      A(    ;
      A     M   1000.5;
      A     DB51.DBX  204.3;
      A     DB51.DBX  203.7;
      AN    DB51.DBX  203.6;
      O     ;
      A     M   1000.6;
      AN    M   1001.0;
      A     M   1100.1;
      O     M   1001.2;
      )     ;
      A     M   1103.1;
      AN    M   1101.7;
      AN    Q    236.6;
      =     Q    236.7;
NETWORK
TITLE =

      A(    ;
      A     M   1000.5;
      A     DB51.DBX  204.4;
      A     DB51.DBX  203.6;
      AN    DB51.DBX  203.7;
      O     ;
      A     M   1000.6;
      AN    M   1001.0;
      A     M   1100.0;
      A     M   5016.0;
      )     ;
      A     M   1103.3;
      AN    M   1102.0;
      AN    Q    237.1;
      =     Q    237.0;
NETWORK
TITLE =

      A(    ;
      A     M   1000.5;
      A     DB51.DBX  204.4;
      A     DB51.DBX  203.7;
      AN    DB51.DBX  203.6;
      O     ;
      A     M   1000.6;
      AN    M   1001.0;
      A     M   1100.1;
      O     M   1001.2;
      )     ;
      A     M   1103.3;
      AN    M   1102.1;
      AN    Q    237.0;
      =     Q    237.1;
NETWORK
TITLE =

      A(    ;
      A     M   1000.5;
      A     DB51.DBX  204.5;
      A     DB51.DBX  203.6;
      AN    DB51.DBX  203.7;
      O     ;
      A     M   1000.6;
      AN    M   1001.0;
      A     M   1100.0;
      A     M   5016.0;
      )     ;
      AN    M   1102.2;
      AN    Q    237.3;
      =     Q    237.2;
NETWORK
TITLE =

      A(    ;
      A     M   1000.5;
      A     DB51.DBX  204.5;
      A     DB51.DBX  203.7;
      AN    DB51.DBX  203.6;
      O     ;
      A     M   1000.6;
      AN    M   1001.0;
      A     M   1100.1;
      A     M   1106.3;
      O     M   1001.2;
      )     ;
      AN    M   1102.3;
      AN    Q    237.2;
      =     Q    237.3;
NETWORK
TITLE =
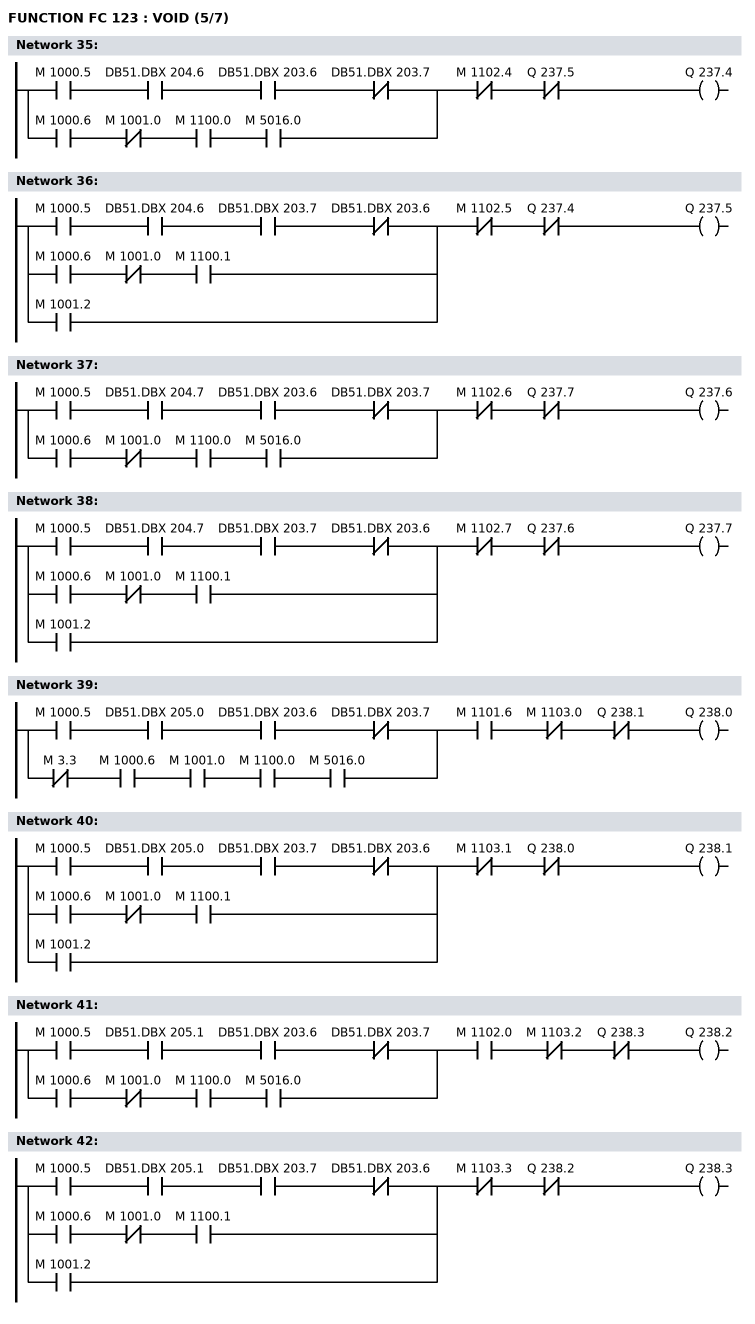

      A(    ;
      A     M   1000.5;
      A     DB51.DBX  204.6;
      A     DB51.DBX  203.6;
      AN    DB51.DBX  203.7;
      O     ;
      A     M   1000.6;
      AN    M   1001.0;
      A     M   1100.0;
      A     M   5016.0;
      )     ;
      AN    M   1102.4;
      AN    Q    237.5;
      =     Q    237.4;
NETWORK
TITLE =

      A(    ;
      A     M   1000.5;
      A     DB51.DBX  204.6;
      A     DB51.DBX  203.7;
      AN    DB51.DBX  203.6;
      O     ;
      A     M   1000.6;
      AN    M   1001.0;
      A     M   1100.1;
      O     M   1001.2;
      )     ;
      AN    M   1102.5;
      AN    Q    237.4;
      =     Q    237.5;
NETWORK
TITLE =

      A(    ;
      A     M   1000.5;
      A     DB51.DBX  204.7;
      A     DB51.DBX  203.6;
      AN    DB51.DBX  203.7;
      O     ;
      A     M   1000.6;
      AN    M   1001.0;
      A     M   1100.0;
      A     M   5016.0;
      )     ;
      AN    M   1102.6;
      AN    Q    237.7;
      =     Q    237.6;
NETWORK
TITLE =

      A(    ;
      A     M   1000.5;
      A     DB51.DBX  204.7;
      A     DB51.DBX  203.7;
      AN    DB51.DBX  203.6;
      O     ;
      A     M   1000.6;
      AN    M   1001.0;
      A     M   1100.1;
      O     M   1001.2;
      )     ;
      AN    M   1102.7;
      AN    Q    237.6;
      =     Q    237.7;
NETWORK
TITLE =

      A(    ;
      A     M   1000.5;
      A     DB51.DBX  205.0;
      A     DB51.DBX  203.6;
      AN    DB51.DBX  203.7;
      O     ;
      AN    M      3.3;
      A     M   1000.6;
      A     M   1001.0;
      A     M   1100.0;
      A     M   5016.0;
      )     ;
      A     M   1101.6;
      AN    M   1103.0;
      AN    Q    238.1;
      =     Q    238.0;
NETWORK
TITLE =

      A(    ;
      A     M   1000.5;
      A     DB51.DBX  205.0;
      A     DB51.DBX  203.7;
      AN    DB51.DBX  203.6;
      O     ;
      A     M   1000.6;
      AN    M   1001.0;
      A     M   1100.1;
      O     M   1001.2;
      )     ;
      AN    M   1103.1;
      AN    Q    238.0;
      =     Q    238.1;
NETWORK
TITLE =

      A(    ;
      A     M   1000.5;
      A     DB51.DBX  205.1;
      A     DB51.DBX  203.6;
      AN    DB51.DBX  203.7;
      O     ;
      A     M   1000.6;
      AN    M   1001.0;
      A     M   1100.0;
      A     M   5016.0;
      )     ;
      A     M   1102.0;
      AN    M   1103.2;
      AN    Q    238.3;
      =     Q    238.2;
NETWORK
TITLE =

      A(    ;
      A     M   1000.5;
      A     DB51.DBX  205.1;
      A     DB51.DBX  203.7;
      AN    DB51.DBX  203.6;
      O     ;
      A     M   1000.6;
      AN    M   1001.0;
      A     M   1100.1;
      O     M   1001.2;
      )     ;
      AN    M   1103.3;
      AN    Q    238.2;
      =     Q    238.3;
NETWORK
TITLE =
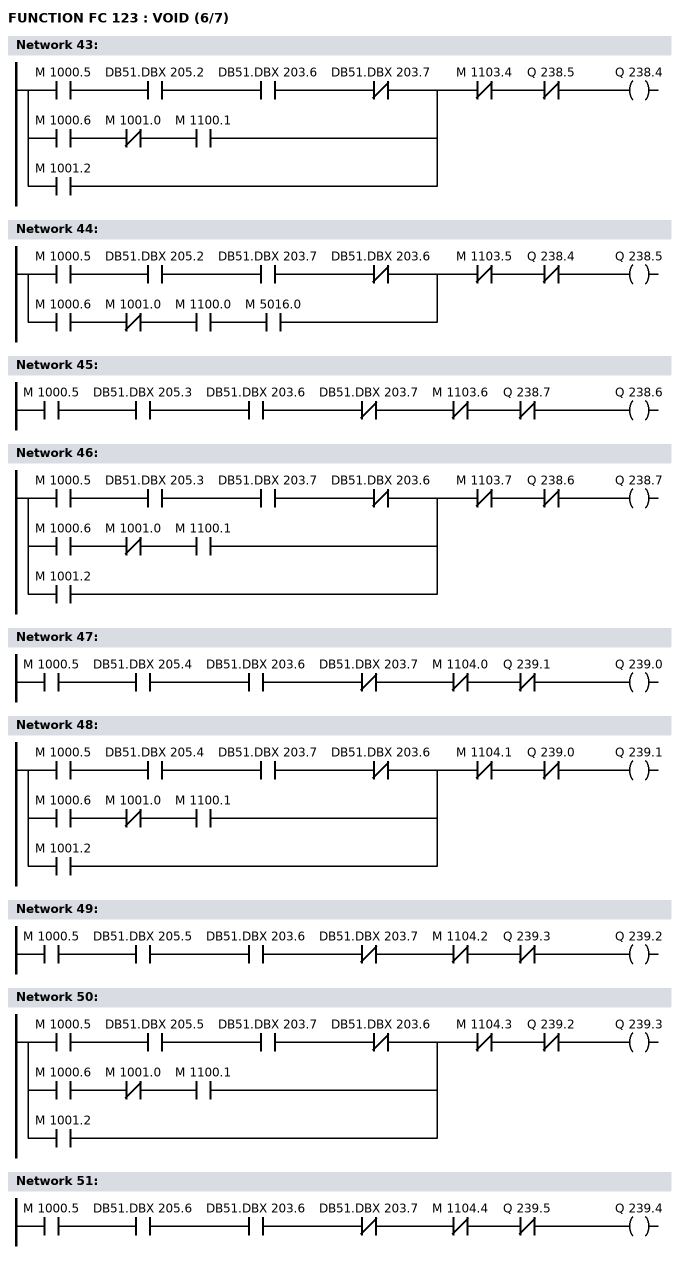

      A(    ;
      A     M   1000.5;
      A     DB51.DBX  205.2;
      A     DB51.DBX  203.6;
      AN    DB51.DBX  203.7;
      O     ;
      A     M   1000.6;
      AN    M   1001.0;
      A     M   1100.1;
      O     M   1001.2;
      )     ;
      AN    M   1103.4;
      AN    Q    238.5;
      =     Q    238.4;
NETWORK
TITLE =

      A(    ;
      A     M   1000.5;
      A     DB51.DBX  205.2;
      A     DB51.DBX  203.7;
      AN    DB51.DBX  203.6;
      O     ;
      A     M   1000.6;
      AN    M   1001.0;
      A     M   1100.0;
      A     M   5016.0;
      )     ;
      AN    M   1103.5;
      AN    Q    238.4;
      =     Q    238.5;
NETWORK
TITLE =

      A     M   1000.5;
      A     DB51.DBX  205.3;
      A     DB51.DBX  203.6;
      AN    DB51.DBX  203.7;
      AN    M   1103.6;
      AN    Q    238.7;
      =     Q    238.6;
NETWORK
TITLE =

      A(    ;
      A     M   1000.5;
      A     DB51.DBX  205.3;
      A     DB51.DBX  203.7;
      AN    DB51.DBX  203.6;
      O     ;
      A     M   1000.6;
      AN    M   1001.0;
      A     M   1100.1;
      O     M   1001.2;
      )     ;
      AN    M   1103.7;
      AN    Q    238.6;
      =     Q    238.7;
NETWORK
TITLE =

      A     M   1000.5;
      A     DB51.DBX  205.4;
      A     DB51.DBX  203.6;
      AN    DB51.DBX  203.7;
      AN    M   1104.0;
      AN    Q    239.1;
      =     Q    239.0;
NETWORK
TITLE =

      A(    ;
      A     M   1000.5;
      A     DB51.DBX  205.4;
      A     DB51.DBX  203.7;
      AN    DB51.DBX  203.6;
      O     ;
      A     M   1000.6;
      AN    M   1001.0;
      A     M   1100.1;
      O     M   1001.2;
      )     ;
      AN    M   1104.1;
      AN    Q    239.0;
      =     Q    239.1;
NETWORK
TITLE =

      A     M   1000.5;
      A     DB51.DBX  205.5;
      A     DB51.DBX  203.6;
      AN    DB51.DBX  203.7;
      AN    M   1104.2;
      AN    Q    239.3;
      =     Q    239.2;
NETWORK
TITLE =

      A(    ;
      A     M   1000.5;
      A     DB51.DBX  205.5;
      A     DB51.DBX  203.7;
      AN    DB51.DBX  203.6;
      O     ;
      A     M   1000.6;
      AN    M   1001.0;
      A     M   1100.1;
      O     M   1001.2;
      )     ;
      AN    M   1104.3;
      AN    Q    239.2;
      =     Q    239.3;
NETWORK
TITLE =

      A     M   1000.5;
      A     DB51.DBX  205.6;
      A     DB51.DBX  203.6;
      AN    DB51.DBX  203.7;
      AN    M   1104.4;
      AN    Q    239.5;
      =     Q    239.4;
NETWORK
TITLE =
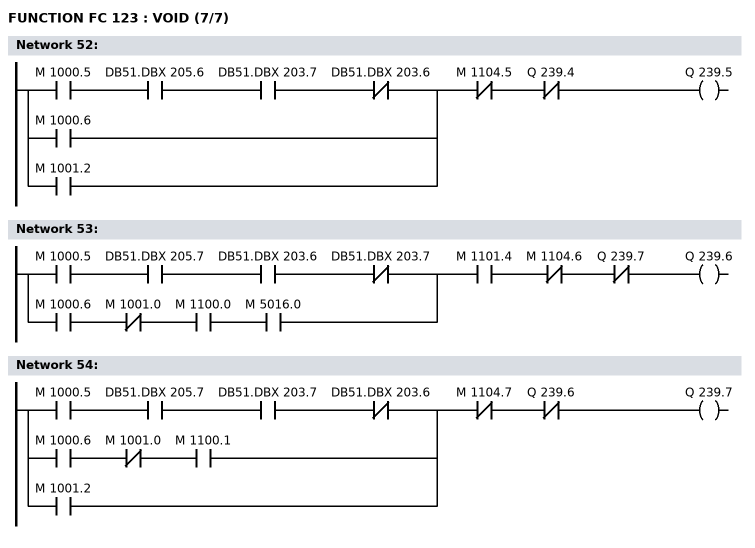

      A(    ;
      A     M   1000.5;
      A     DB51.DBX  205.6;
      A     DB51.DBX  203.7;
      AN    DB51.DBX  203.6;
      O     M   1000.6;
      O     M   1001.2;
      )     ;
      AN    M   1104.5;
      AN    Q    239.4;
      =     Q    239.5;
NETWORK
TITLE =

      A(    ;
      A     M   1000.5;
      A     DB51.DBX  205.7;
      A     DB51.DBX  203.6;
      AN    DB51.DBX  203.7;
      O     ;
      A     M   1000.6;
      AN    M   1001.0;
      A     M   1100.0;
      A     M   5016.0;
      )     ;
      A     M   1101.4;
      AN    M   1104.6;
      AN    Q    239.7;
      =     Q    239.6;
NETWORK
TITLE =

      A(    ;
      A     M   1000.5;
      A     DB51.DBX  205.7;
      A     DB51.DBX  203.7;
      AN    DB51.DBX  203.6;
      O     ;
      A     M   1000.6;
      AN    M   1001.0;
      A     M   1100.1;
      O     M   1001.2;
      )     ;
      AN    M   1104.7;
      AN    Q    239.6;
      =     Q    239.7;
END_FUNCTION

FUNCTION_BLOCK FB 124
TITLE =
VERSION : 0.1


VAR
  S702_TL_DC_PIN : FB 426;
  S702_TL_DC_LATCH1 : FB 426;
  S702_TL_DC_LATCH2 : FB 426;
  S702_TL_DC_1ST_CLAMP1 : FB 426;
  S702_TL_DC_1ST_CLAMP2 : FB 426;
  S702_TL_DC_1ST_CLAMP3 : FB 426;
  S702_TL_DC_2ND_CLAMP1 : FB 426;
  S702_TL_DC_2ND_CLAMP2 : FB 426;
  S702_TL_DC_U261 : FB 426;
  S702_TL_DC_U261_CLAMP : FB 426;
  S702_TL_DC_U269 : FB 426;
  S702_TL_DC_U269_CLAMP : FB 426;
  S702_TL_DC_3RD_CLAMP : FB 426;
  S702_TL_DC_U262_1_UP_DN : FB 426;
  S702_TL_DC_U262_1 : FB 426;
  S702_TL_DC_U262_1_CLAMP : FB 426;
  S702_TL_DC_U261_2_CLAMP : FB 426;
END_VAR
BEGIN
NETWORK
TITLE =
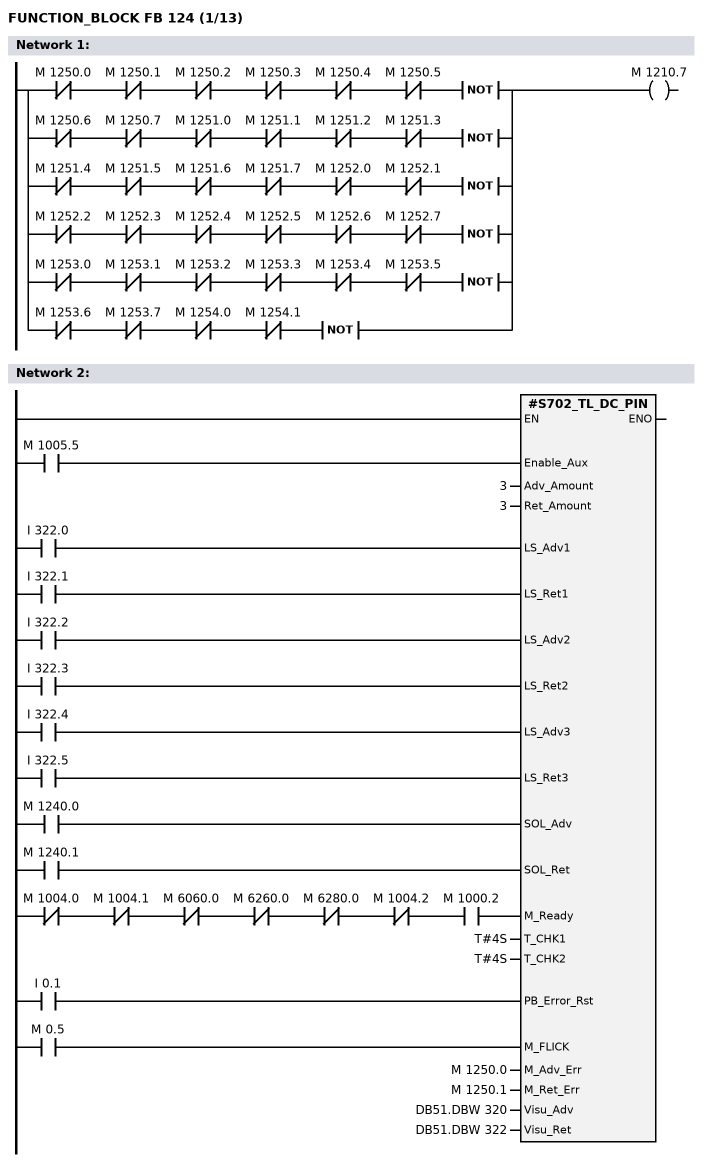

      AN    M   1250.0;
      AN    M   1250.1;
      AN    M   1250.2;
      AN    M   1250.3;
      AN    M   1250.4;
      AN    M   1250.5;
      NOT   ;
      O(    ;
      AN    M   1250.6;
      AN    M   1250.7;
      AN    M   1251.0;
      AN    M   1251.1;
      AN    M   1251.2;
      AN    M   1251.3;
      NOT   ;
      )     ;
      O(    ;
      AN    M   1251.4;
      AN    M   1251.5;
      AN    M   1251.6;
      AN    M   1251.7;
      AN    M   1252.0;
      AN    M   1252.1;
      NOT   ;
      )     ;
      O(    ;
      AN    M   1252.2;
      AN    M   1252.3;
      AN    M   1252.4;
      AN    M   1252.5;
      AN    M   1252.6;
      AN    M   1252.7;
      NOT   ;
      )     ;
      O(    ;
      AN    M   1253.0;
      AN    M   1253.1;
      AN    M   1253.2;
      AN    M   1253.3;
      AN    M   1253.4;
      AN    M   1253.5;
      NOT   ;
      )     ;
      O(    ;
      AN    M   1253.6;
      AN    M   1253.7;
      AN    M   1254.0;
      AN    M   1254.1;
      NOT   ;
      )     ;
      =     M   1210.7;
NETWORK
TITLE =

      A     M   1005.5;
      =     L      0.0;
      BLD   103;
      A     I    322.0;
      =     L      0.1;
      BLD   103;
      A     I    322.1;
      =     L      0.2;
      BLD   103;
      A     I    322.2;
      =     L      0.3;
      BLD   103;
      A     I    322.3;
      =     L      0.4;
      BLD   103;
      A     I    322.4;
      =     L      0.5;
      BLD   103;
      A     I    322.5;
      =     L      0.6;
      BLD   103;
      A     M   1240.0;
      =     L      2.1;
      BLD   103;
      A     M   1240.1;
      =     L      2.2;
      BLD   103;
      AN    M   1004.0;
      AN    M   1004.1;
      AN    M   6060.0;
      AN    M   6260.0;
      AN    M   6280.0;
      AN    M   1004.2;
      A     M   1000.2;
      =     L      2.3;
      BLD   103;
      A     I      0.1;
      =     L      2.5;
      BLD   103;
      A     M      0.5;
      =     L      2.6;
      BLD   103;
      CALL #S702_TL_DC_PIN (
           Enable_Aux               := L      0.0,
           Adv_Amount               := 3,
           Ret_Amount               := 3,
           LS_Adv1                  := L      0.1,
           LS_Ret1                  := L      0.2,
           LS_Adv2                  := L      0.3,
           LS_Ret2                  := L      0.4,
           LS_Adv3                  := L      0.5,
           LS_Ret3                  := L      0.6,
           SOL_Adv                  := L      2.1,
           SOL_Ret                  := L      2.2,
           M_Ready                  := L      2.3,
           T_CHK1                   := T#4S,
           T_CHK2                   := T#4S,
           PB_Error_Rst             := L      2.5,
           M_FLICK                  := L      2.6,
           M_Adv_Err                := M   1250.0,
           M_Ret_Err                := M   1250.1,
           Visu_Adv                 := DB51.DBW  320,
           Visu_Ret                 := DB51.DBW  322);
      NOP   0;
NETWORK
TITLE =
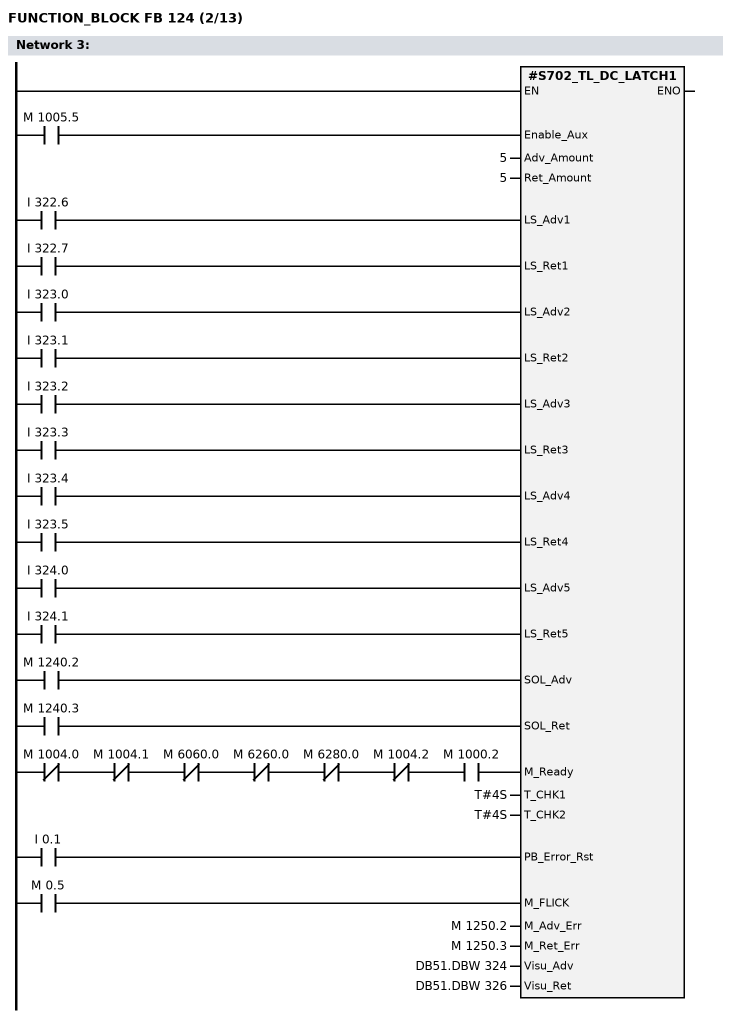

      A     M   1005.5;
      =     L      0.0;
      BLD   103;
      A     I    322.6;
      =     L      0.1;
      BLD   103;
      A     I    322.7;
      =     L      0.2;
      BLD   103;
      A     I    323.0;
      =     L      0.3;
      BLD   103;
      A     I    323.1;
      =     L      0.4;
      BLD   103;
      A     I    323.2;
      =     L      0.5;
      BLD   103;
      A     I    323.3;
      =     L      0.6;
      BLD   103;
      A     I    323.4;
      =     L      0.7;
      BLD   103;
      A     I    323.5;
      =     L      1.0;
      BLD   103;
      A     I    324.0;
      =     L      1.1;
      BLD   103;
      A     I    324.1;
      =     L      1.2;
      BLD   103;
      A     M   1240.2;
      =     L      2.1;
      BLD   103;
      A     M   1240.3;
      =     L      2.2;
      BLD   103;
      AN    M   1004.0;
      AN    M   1004.1;
      AN    M   6060.0;
      AN    M   6260.0;
      AN    M   6280.0;
      AN    M   1004.2;
      A     M   1000.2;
      =     L      2.3;
      BLD   103;
      A     I      0.1;
      =     L      2.5;
      BLD   103;
      A     M      0.5;
      =     L      2.6;
      BLD   103;
      CALL #S702_TL_DC_LATCH1 (
           Enable_Aux               := L      0.0,
           Adv_Amount               := 5,
           Ret_Amount               := 5,
           LS_Adv1                  := L      0.1,
           LS_Ret1                  := L      0.2,
           LS_Adv2                  := L      0.3,
           LS_Ret2                  := L      0.4,
           LS_Adv3                  := L      0.5,
           LS_Ret3                  := L      0.6,
           LS_Adv4                  := L      0.7,
           LS_Ret4                  := L      1.0,
           LS_Adv5                  := L      1.1,
           LS_Ret5                  := L      1.2,
           SOL_Adv                  := L      2.1,
           SOL_Ret                  := L      2.2,
           M_Ready                  := L      2.3,
           T_CHK1                   := T#4S,
           T_CHK2                   := T#4S,
           PB_Error_Rst             := L      2.5,
           M_FLICK                  := L      2.6,
           M_Adv_Err                := M   1250.2,
           M_Ret_Err                := M   1250.3,
           Visu_Adv                 := DB51.DBW  324,
           Visu_Ret                 := DB51.DBW  326);
      NOP   0;
NETWORK
TITLE =
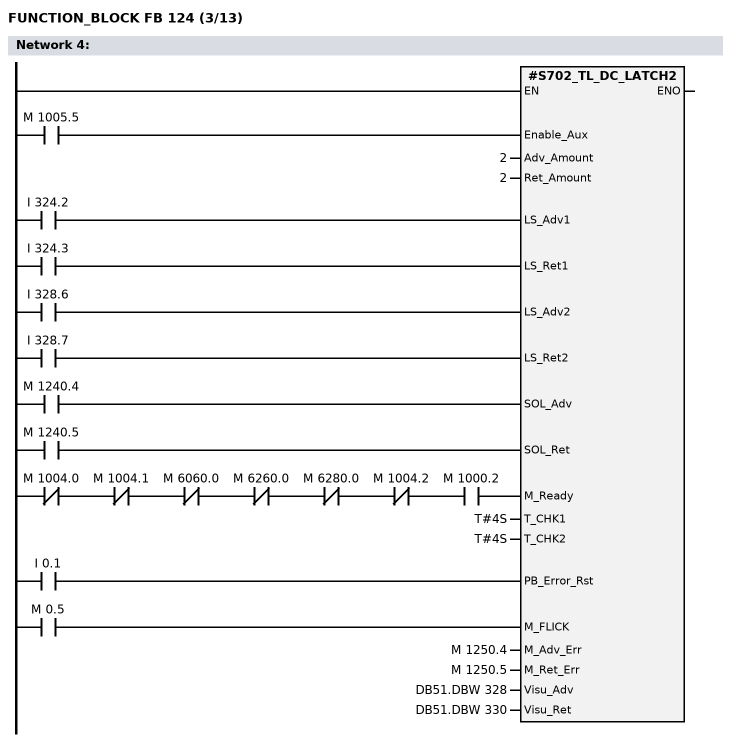

      A     M   1005.5;
      =     L      0.0;
      BLD   103;
      A     I    324.2;
      =     L      0.1;
      BLD   103;
      A     I    324.3;
      =     L      0.2;
      BLD   103;
      A     I    328.6;
      =     L      0.3;
      BLD   103;
      A     I    328.7;
      =     L      0.4;
      BLD   103;
      A     M   1240.4;
      =     L      2.1;
      BLD   103;
      A     M   1240.5;
      =     L      2.2;
      BLD   103;
      AN    M   1004.0;
      AN    M   1004.1;
      AN    M   6060.0;
      AN    M   6260.0;
      AN    M   6280.0;
      AN    M   1004.2;
      A     M   1000.2;
      =     L      2.3;
      BLD   103;
      A     I      0.1;
      =     L      2.5;
      BLD   103;
      A     M      0.5;
      =     L      2.6;
      BLD   103;
      CALL #S702_TL_DC_LATCH2 (
           Enable_Aux               := L      0.0,
           Adv_Amount               := 2,
           Ret_Amount               := 2,
           LS_Adv1                  := L      0.1,
           LS_Ret1                  := L      0.2,
           LS_Adv2                  := L      0.3,
           LS_Ret2                  := L      0.4,
           SOL_Adv                  := L      2.1,
           SOL_Ret                  := L      2.2,
           M_Ready                  := L      2.3,
           T_CHK1                   := T#4S,
           T_CHK2                   := T#4S,
           PB_Error_Rst             := L      2.5,
           M_FLICK                  := L      2.6,
           M_Adv_Err                := M   1250.4,
           M_Ret_Err                := M   1250.5,
           Visu_Adv                 := DB51.DBW  328,
           Visu_Ret                 := DB51.DBW  330);
      NOP   0;
NETWORK
TITLE =
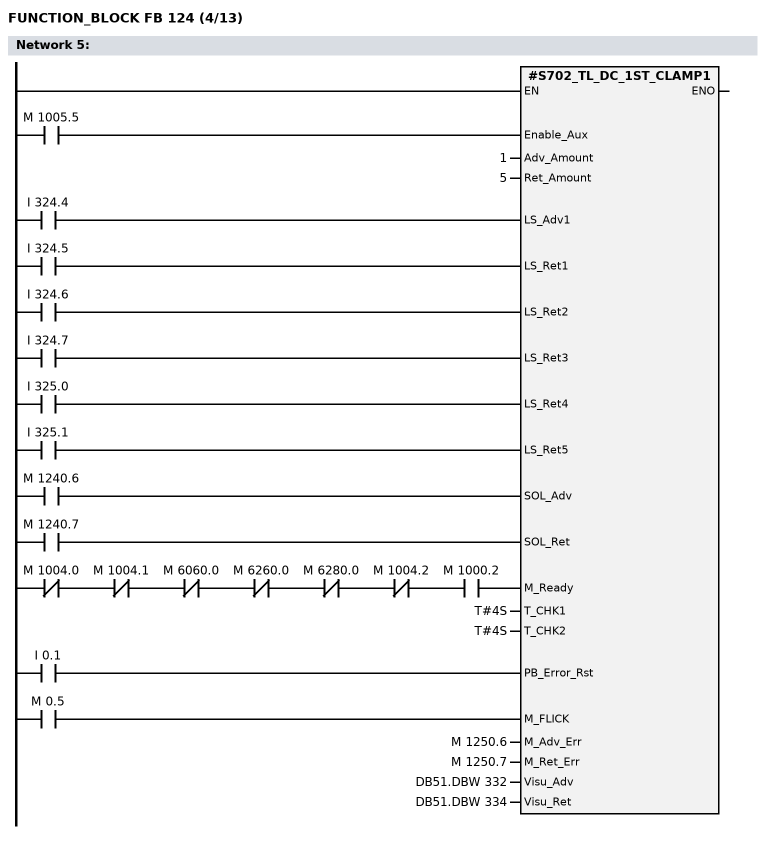

      A     M   1005.5;
      =     L      0.0;
      BLD   103;
      A     I    324.4;
      =     L      0.1;
      BLD   103;
      A     I    324.5;
      =     L      0.2;
      BLD   103;
      A     I    324.6;
      =     L      0.4;
      BLD   103;
      A     I    324.7;
      =     L      0.6;
      BLD   103;
      A     I    325.0;
      =     L      1.0;
      BLD   103;
      A     I    325.1;
      =     L      1.2;
      BLD   103;
      A     M   1240.6;
      =     L      2.1;
      BLD   103;
      A     M   1240.7;
      =     L      2.2;
      BLD   103;
      AN    M   1004.0;
      AN    M   1004.1;
      AN    M   6060.0;
      AN    M   6260.0;
      AN    M   6280.0;
      AN    M   1004.2;
      A     M   1000.2;
      =     L      2.3;
      BLD   103;
      A     I      0.1;
      =     L      2.5;
      BLD   103;
      A     M      0.5;
      =     L      2.6;
      BLD   103;
      CALL #S702_TL_DC_1ST_CLAMP1 (
           Enable_Aux               := L      0.0,
           Adv_Amount               := 1,
           Ret_Amount               := 5,
           LS_Adv1                  := L      0.1,
           LS_Ret1                  := L      0.2,
           LS_Ret2                  := L      0.4,
           LS_Ret3                  := L      0.6,
           LS_Ret4                  := L      1.0,
           LS_Ret5                  := L      1.2,
           SOL_Adv                  := L      2.1,
           SOL_Ret                  := L      2.2,
           M_Ready                  := L      2.3,
           T_CHK1                   := T#4S,
           T_CHK2                   := T#4S,
           PB_Error_Rst             := L      2.5,
           M_FLICK                  := L      2.6,
           M_Adv_Err                := M   1250.6,
           M_Ret_Err                := M   1250.7,
           Visu_Adv                 := DB51.DBW  332,
           Visu_Ret                 := DB51.DBW  334);
      NOP   0;
NETWORK
TITLE =
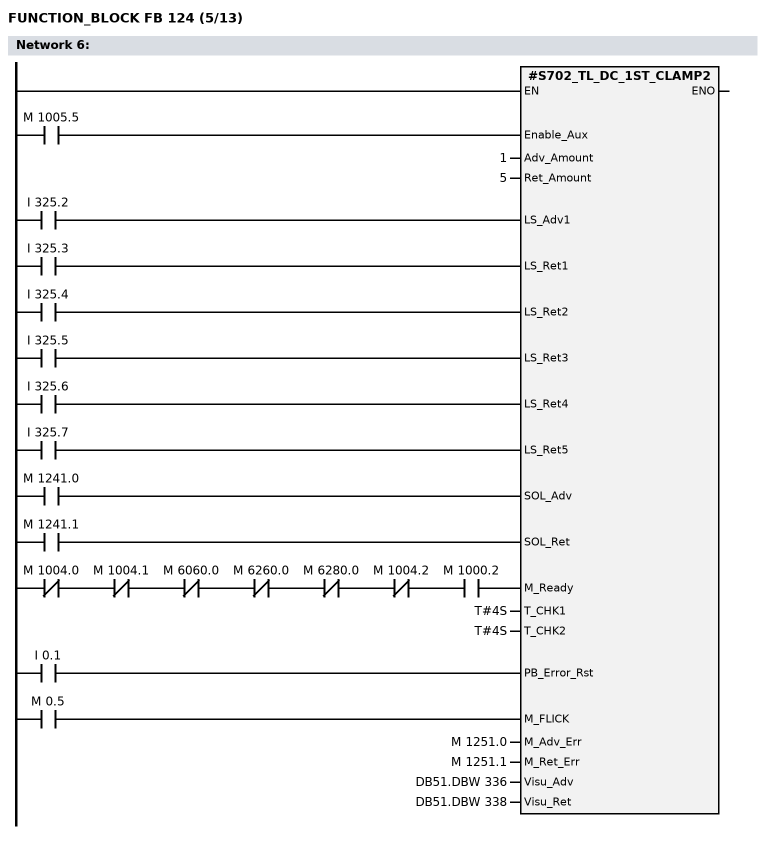

      A     M   1005.5;
      =     L      0.0;
      BLD   103;
      A     I    325.2;
      =     L      0.1;
      BLD   103;
      A     I    325.3;
      =     L      0.2;
      BLD   103;
      A     I    325.4;
      =     L      0.4;
      BLD   103;
      A     I    325.5;
      =     L      0.6;
      BLD   103;
      A     I    325.6;
      =     L      1.0;
      BLD   103;
      A     I    325.7;
      =     L      1.2;
      BLD   103;
      A     M   1241.0;
      =     L      2.1;
      BLD   103;
      A     M   1241.1;
      =     L      2.2;
      BLD   103;
      AN    M   1004.0;
      AN    M   1004.1;
      AN    M   6060.0;
      AN    M   6260.0;
      AN    M   6280.0;
      AN    M   1004.2;
      A     M   1000.2;
      =     L      2.3;
      BLD   103;
      A     I      0.1;
      =     L      2.5;
      BLD   103;
      A     M      0.5;
      =     L      2.6;
      BLD   103;
      CALL #S702_TL_DC_1ST_CLAMP2 (
           Enable_Aux               := L      0.0,
           Adv_Amount               := 1,
           Ret_Amount               := 5,
           LS_Adv1                  := L      0.1,
           LS_Ret1                  := L      0.2,
           LS_Ret2                  := L      0.4,
           LS_Ret3                  := L      0.6,
           LS_Ret4                  := L      1.0,
           LS_Ret5                  := L      1.2,
           SOL_Adv                  := L      2.1,
           SOL_Ret                  := L      2.2,
           M_Ready                  := L      2.3,
           T_CHK1                   := T#4S,
           T_CHK2                   := T#4S,
           PB_Error_Rst             := L      2.5,
           M_FLICK                  := L      2.6,
           M_Adv_Err                := M   1251.0,
           M_Ret_Err                := M   1251.1,
           Visu_Adv                 := DB51.DBW  336,
           Visu_Ret                 := DB51.DBW  338);
      NOP   0;
NETWORK
TITLE =
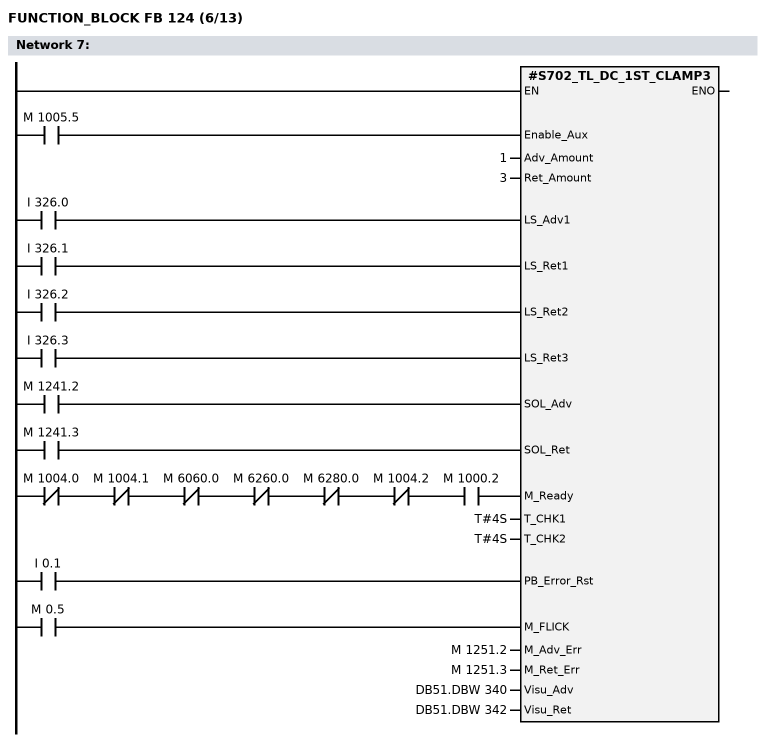

      A     M   1005.5;
      =     L      0.0;
      BLD   103;
      A     I    326.0;
      =     L      0.1;
      BLD   103;
      A     I    326.1;
      =     L      0.2;
      BLD   103;
      A     I    326.2;
      =     L      0.4;
      BLD   103;
      A     I    326.3;
      =     L      0.6;
      BLD   103;
      A     M   1241.2;
      =     L      2.1;
      BLD   103;
      A     M   1241.3;
      =     L      2.2;
      BLD   103;
      AN    M   1004.0;
      AN    M   1004.1;
      AN    M   6060.0;
      AN    M   6260.0;
      AN    M   6280.0;
      AN    M   1004.2;
      A     M   1000.2;
      =     L      2.3;
      BLD   103;
      A     I      0.1;
      =     L      2.5;
      BLD   103;
      A     M      0.5;
      =     L      2.6;
      BLD   103;
      CALL #S702_TL_DC_1ST_CLAMP3 (
           Enable_Aux               := L      0.0,
           Adv_Amount               := 1,
           Ret_Amount               := 3,
           LS_Adv1                  := L      0.1,
           LS_Ret1                  := L      0.2,
           LS_Ret2                  := L      0.4,
           LS_Ret3                  := L      0.6,
           SOL_Adv                  := L      2.1,
           SOL_Ret                  := L      2.2,
           M_Ready                  := L      2.3,
           T_CHK1                   := T#4S,
           T_CHK2                   := T#4S,
           PB_Error_Rst             := L      2.5,
           M_FLICK                  := L      2.6,
           M_Adv_Err                := M   1251.2,
           M_Ret_Err                := M   1251.3,
           Visu_Adv                 := DB51.DBW  340,
           Visu_Ret                 := DB51.DBW  342);
      NOP   0;
NETWORK
TITLE =
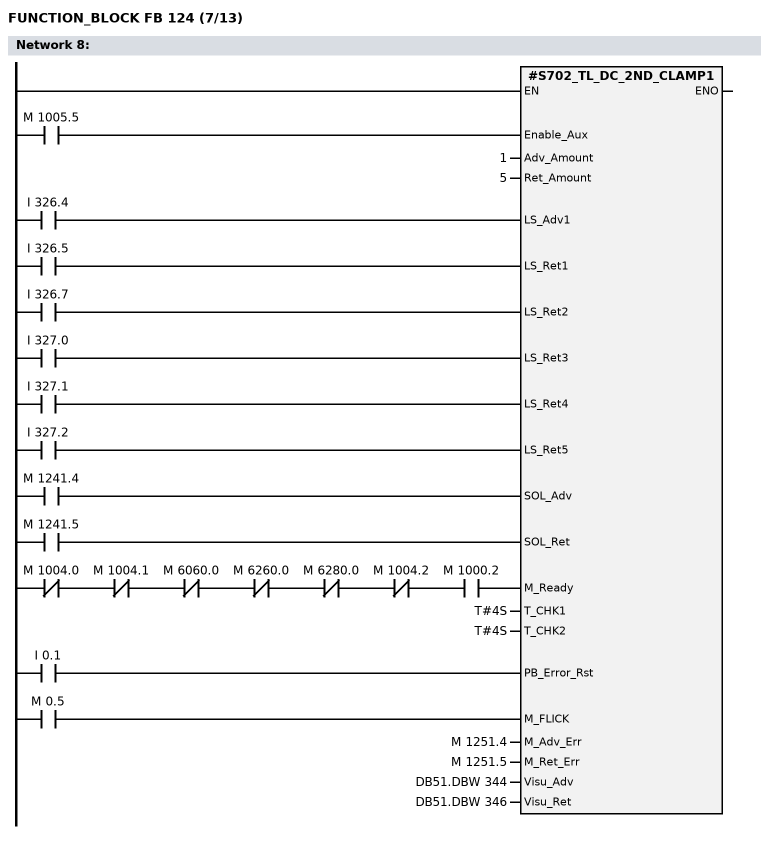

      A     M   1005.5;
      =     L      0.0;
      BLD   103;
      A     I    326.4;
      =     L      0.1;
      BLD   103;
      A     I    326.5;
      =     L      0.2;
      BLD   103;
      A     I    326.7;
      =     L      0.4;
      BLD   103;
      A     I    327.0;
      =     L      0.6;
      BLD   103;
      A     I    327.1;
      =     L      1.0;
      BLD   103;
      A     I    327.2;
      =     L      1.2;
      BLD   103;
      A     M   1241.4;
      =     L      2.1;
      BLD   103;
      A     M   1241.5;
      =     L      2.2;
      BLD   103;
      AN    M   1004.0;
      AN    M   1004.1;
      AN    M   6060.0;
      AN    M   6260.0;
      AN    M   6280.0;
      AN    M   1004.2;
      A     M   1000.2;
      =     L      2.3;
      BLD   103;
      A     I      0.1;
      =     L      2.5;
      BLD   103;
      A     M      0.5;
      =     L      2.6;
      BLD   103;
      CALL #S702_TL_DC_2ND_CLAMP1 (
           Enable_Aux               := L      0.0,
           Adv_Amount               := 1,
           Ret_Amount               := 5,
           LS_Adv1                  := L      0.1,
           LS_Ret1                  := L      0.2,
           LS_Ret2                  := L      0.4,
           LS_Ret3                  := L      0.6,
           LS_Ret4                  := L      1.0,
           LS_Ret5                  := L      1.2,
           SOL_Adv                  := L      2.1,
           SOL_Ret                  := L      2.2,
           M_Ready                  := L      2.3,
           T_CHK1                   := T#4S,
           T_CHK2                   := T#4S,
           PB_Error_Rst             := L      2.5,
           M_FLICK                  := L      2.6,
           M_Adv_Err                := M   1251.4,
           M_Ret_Err                := M   1251.5,
           Visu_Adv                 := DB51.DBW  344,
           Visu_Ret                 := DB51.DBW  346);
      NOP   0;
NETWORK
TITLE =
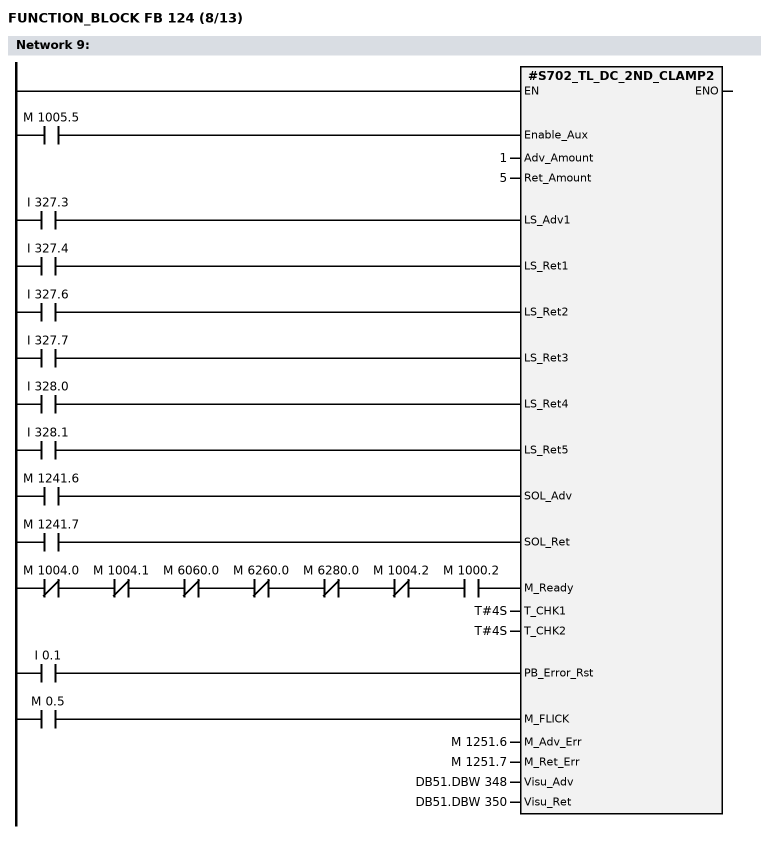

      A     M   1005.5;
      =     L      0.0;
      BLD   103;
      A     I    327.3;
      =     L      0.1;
      BLD   103;
      A     I    327.4;
      =     L      0.2;
      BLD   103;
      A     I    327.6;
      =     L      0.4;
      BLD   103;
      A     I    327.7;
      =     L      0.6;
      BLD   103;
      A     I    328.0;
      =     L      1.0;
      BLD   103;
      A     I    328.1;
      =     L      1.2;
      BLD   103;
      A     M   1241.6;
      =     L      2.1;
      BLD   103;
      A     M   1241.7;
      =     L      2.2;
      BLD   103;
      AN    M   1004.0;
      AN    M   1004.1;
      AN    M   6060.0;
      AN    M   6260.0;
      AN    M   6280.0;
      AN    M   1004.2;
      A     M   1000.2;
      =     L      2.3;
      BLD   103;
      A     I      0.1;
      =     L      2.5;
      BLD   103;
      A     M      0.5;
      =     L      2.6;
      BLD   103;
      CALL #S702_TL_DC_2ND_CLAMP2 (
           Enable_Aux               := L      0.0,
           Adv_Amount               := 1,
           Ret_Amount               := 5,
           LS_Adv1                  := L      0.1,
           LS_Ret1                  := L      0.2,
           LS_Ret2                  := L      0.4,
           LS_Ret3                  := L      0.6,
           LS_Ret4                  := L      1.0,
           LS_Ret5                  := L      1.2,
           SOL_Adv                  := L      2.1,
           SOL_Ret                  := L      2.2,
           M_Ready                  := L      2.3,
           T_CHK1                   := T#4S,
           T_CHK2                   := T#4S,
           PB_Error_Rst             := L      2.5,
           M_FLICK                  := L      2.6,
           M_Adv_Err                := M   1251.6,
           M_Ret_Err                := M   1251.7,
           Visu_Adv                 := DB51.DBW  348,
           Visu_Ret                 := DB51.DBW  350);
      NOP   0;
NETWORK
TITLE =
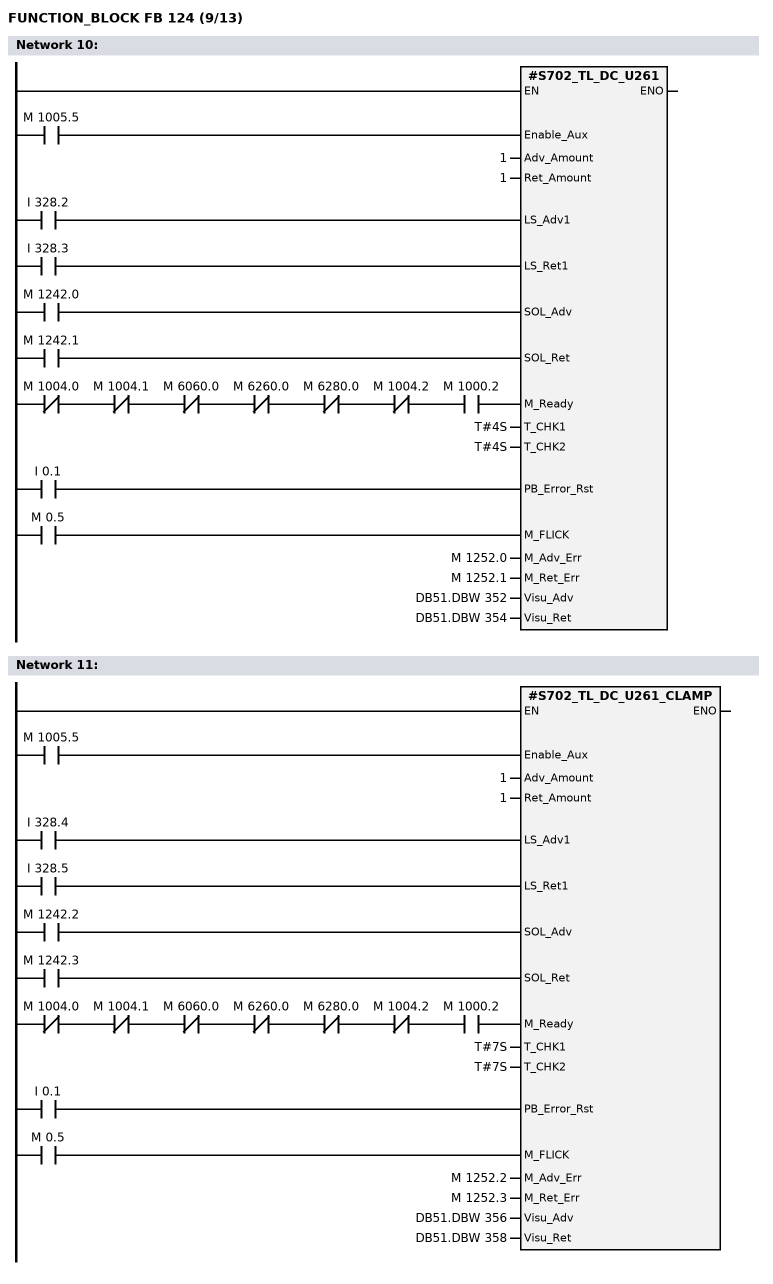

      A     M   1005.5;
      =     L      0.0;
      BLD   103;
      A     I    328.2;
      =     L      0.1;
      BLD   103;
      A     I    328.3;
      =     L      0.2;
      BLD   103;
      A     M   1242.0;
      =     L      2.1;
      BLD   103;
      A     M   1242.1;
      =     L      2.2;
      BLD   103;
      AN    M   1004.0;
      AN    M   1004.1;
      AN    M   6060.0;
      AN    M   6260.0;
      AN    M   6280.0;
      AN    M   1004.2;
      A     M   1000.2;
      =     L      2.3;
      BLD   103;
      A     I      0.1;
      =     L      2.5;
      BLD   103;
      A     M      0.5;
      =     L      2.6;
      BLD   103;
      CALL #S702_TL_DC_U261 (
           Enable_Aux               := L      0.0,
           Adv_Amount               := 1,
           Ret_Amount               := 1,
           LS_Adv1                  := L      0.1,
           LS_Ret1                  := L      0.2,
           SOL_Adv                  := L      2.1,
           SOL_Ret                  := L      2.2,
           M_Ready                  := L      2.3,
           T_CHK1                   := T#4S,
           T_CHK2                   := T#4S,
           PB_Error_Rst             := L      2.5,
           M_FLICK                  := L      2.6,
           M_Adv_Err                := M   1252.0,
           M_Ret_Err                := M   1252.1,
           Visu_Adv                 := DB51.DBW  352,
           Visu_Ret                 := DB51.DBW  354);
      NOP   0;
NETWORK
TITLE =

      A     M   1005.5;
      =     L      0.0;
      BLD   103;
      A     I    328.4;
      =     L      0.1;
      BLD   103;
      A     I    328.5;
      =     L      0.2;
      BLD   103;
      A     M   1242.2;
      =     L      2.1;
      BLD   103;
      A     M   1242.3;
      =     L      2.2;
      BLD   103;
      AN    M   1004.0;
      AN    M   1004.1;
      AN    M   6060.0;
      AN    M   6260.0;
      AN    M   6280.0;
      AN    M   1004.2;
      A     M   1000.2;
      =     L      2.3;
      BLD   103;
      A     I      0.1;
      =     L      2.5;
      BLD   103;
      A     M      0.5;
      =     L      2.6;
      BLD   103;
      CALL #S702_TL_DC_U261_CLAMP (
           Enable_Aux               := L      0.0,
           Adv_Amount               := 1,
           Ret_Amount               := 1,
           LS_Adv1                  := L      0.1,
           LS_Ret1                  := L      0.2,
           SOL_Adv                  := L      2.1,
           SOL_Ret                  := L      2.2,
           M_Ready                  := L      2.3,
           T_CHK1                   := T#7S,
           T_CHK2                   := T#7S,
           PB_Error_Rst             := L      2.5,
           M_FLICK                  := L      2.6,
           M_Adv_Err                := M   1252.2,
           M_Ret_Err                := M   1252.3,
           Visu_Adv                 := DB51.DBW  356,
           Visu_Ret                 := DB51.DBW  358);
      NOP   0;
NETWORK
TITLE =
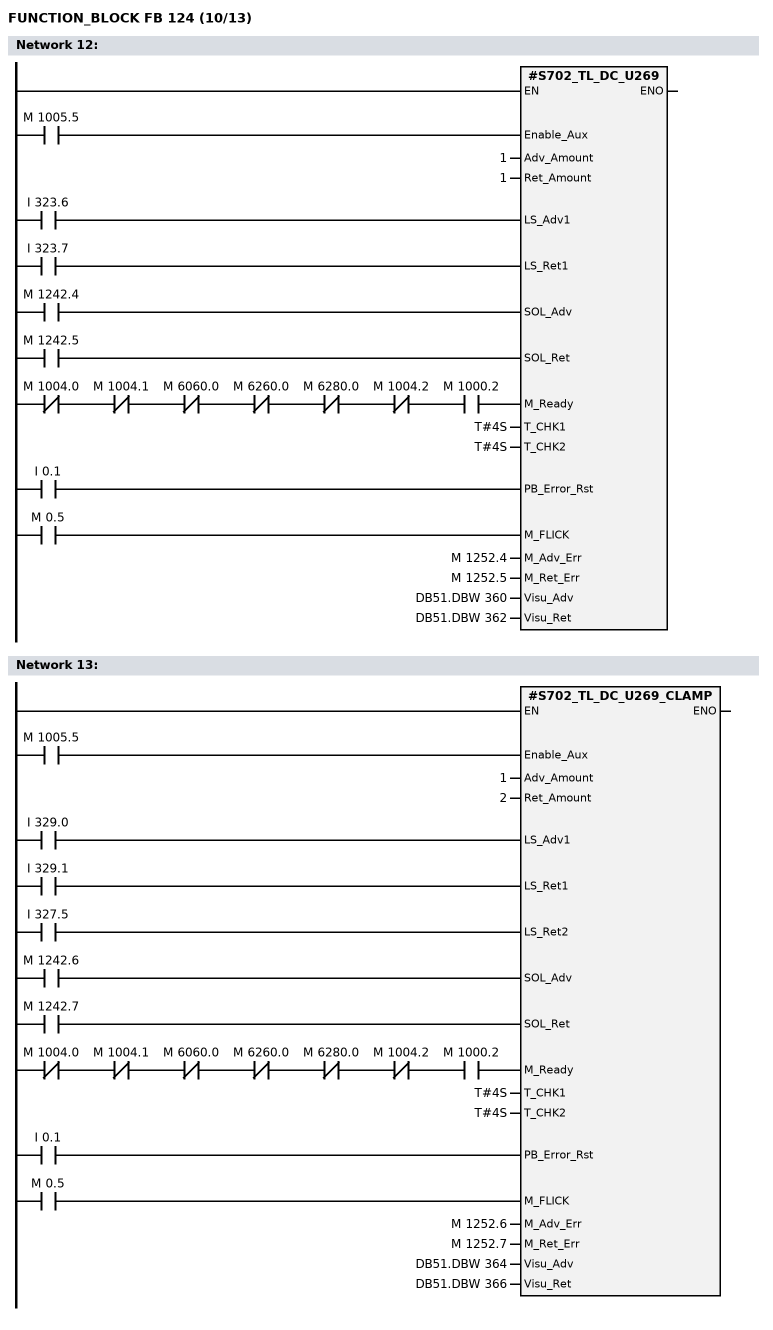

      A     M   1005.5;
      =     L      0.0;
      BLD   103;
      A     I    323.6;
      =     L      0.1;
      BLD   103;
      A     I    323.7;
      =     L      0.2;
      BLD   103;
      A     M   1242.4;
      =     L      2.1;
      BLD   103;
      A     M   1242.5;
      =     L      2.2;
      BLD   103;
      AN    M   1004.0;
      AN    M   1004.1;
      AN    M   6060.0;
      AN    M   6260.0;
      AN    M   6280.0;
      AN    M   1004.2;
      A     M   1000.2;
      =     L      2.3;
      BLD   103;
      A     I      0.1;
      =     L      2.5;
      BLD   103;
      A     M      0.5;
      =     L      2.6;
      BLD   103;
      CALL #S702_TL_DC_U269 (
           Enable_Aux               := L      0.0,
           Adv_Amount               := 1,
           Ret_Amount               := 1,
           LS_Adv1                  := L      0.1,
           LS_Ret1                  := L      0.2,
           SOL_Adv                  := L      2.1,
           SOL_Ret                  := L      2.2,
           M_Ready                  := L      2.3,
           T_CHK1                   := T#4S,
           T_CHK2                   := T#4S,
           PB_Error_Rst             := L      2.5,
           M_FLICK                  := L      2.6,
           M_Adv_Err                := M   1252.4,
           M_Ret_Err                := M   1252.5,
           Visu_Adv                 := DB51.DBW  360,
           Visu_Ret                 := DB51.DBW  362);
      NOP   0;
NETWORK
TITLE =

      A     M   1005.5;
      =     L      0.0;
      BLD   103;
      A     I    329.0;
      =     L      0.1;
      BLD   103;
      A     I    329.1;
      =     L      0.2;
      BLD   103;
      A     I    327.5;
      =     L      0.4;
      BLD   103;
      A     M   1242.6;
      =     L      2.1;
      BLD   103;
      A     M   1242.7;
      =     L      2.2;
      BLD   103;
      AN    M   1004.0;
      AN    M   1004.1;
      AN    M   6060.0;
      AN    M   6260.0;
      AN    M   6280.0;
      AN    M   1004.2;
      A     M   1000.2;
      =     L      2.3;
      BLD   103;
      A     I      0.1;
      =     L      2.5;
      BLD   103;
      A     M      0.5;
      =     L      2.6;
      BLD   103;
      CALL #S702_TL_DC_U269_CLAMP (
           Enable_Aux               := L      0.0,
           Adv_Amount               := 1,
           Ret_Amount               := 2,
           LS_Adv1                  := L      0.1,
           LS_Ret1                  := L      0.2,
           LS_Ret2                  := L      0.4,
           SOL_Adv                  := L      2.1,
           SOL_Ret                  := L      2.2,
           M_Ready                  := L      2.3,
           T_CHK1                   := T#4S,
           T_CHK2                   := T#4S,
           PB_Error_Rst             := L      2.5,
           M_FLICK                  := L      2.6,
           M_Adv_Err                := M   1252.6,
           M_Ret_Err                := M   1252.7,
           Visu_Adv                 := DB51.DBW  364,
           Visu_Ret                 := DB51.DBW  366);
      NOP   0;
NETWORK
TITLE =
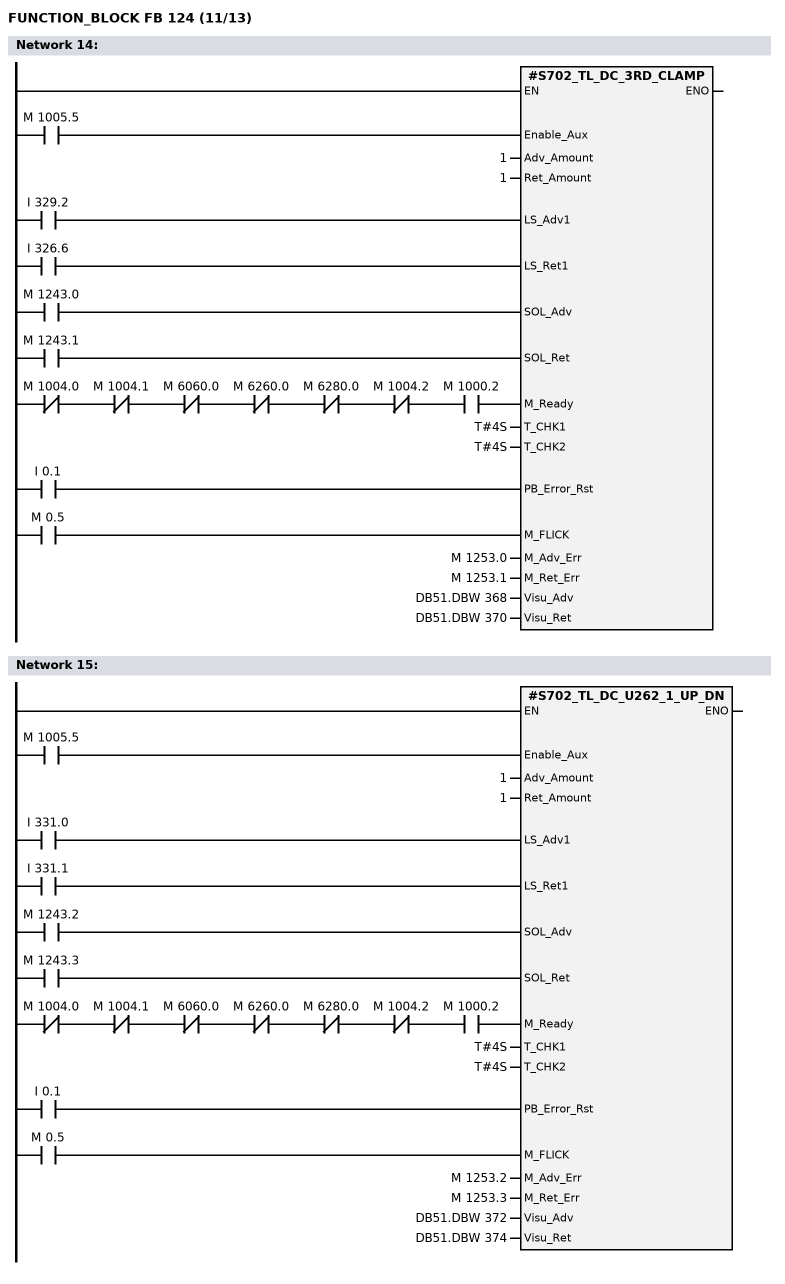

      A     M   1005.5;
      =     L      0.0;
      BLD   103;
      A     I    329.2;
      =     L      0.1;
      BLD   103;
      A     I    326.6;
      =     L      0.2;
      BLD   103;
      A     M   1243.0;
      =     L      2.1;
      BLD   103;
      A     M   1243.1;
      =     L      2.2;
      BLD   103;
      AN    M   1004.0;
      AN    M   1004.1;
      AN    M   6060.0;
      AN    M   6260.0;
      AN    M   6280.0;
      AN    M   1004.2;
      A     M   1000.2;
      =     L      2.3;
      BLD   103;
      A     I      0.1;
      =     L      2.5;
      BLD   103;
      A     M      0.5;
      =     L      2.6;
      BLD   103;
      CALL #S702_TL_DC_3RD_CLAMP (
           Enable_Aux               := L      0.0,
           Adv_Amount               := 1,
           Ret_Amount               := 1,
           LS_Adv1                  := L      0.1,
           LS_Ret1                  := L      0.2,
           SOL_Adv                  := L      2.1,
           SOL_Ret                  := L      2.2,
           M_Ready                  := L      2.3,
           T_CHK1                   := T#4S,
           T_CHK2                   := T#4S,
           PB_Error_Rst             := L      2.5,
           M_FLICK                  := L      2.6,
           M_Adv_Err                := M   1253.0,
           M_Ret_Err                := M   1253.1,
           Visu_Adv                 := DB51.DBW  368,
           Visu_Ret                 := DB51.DBW  370);
      NOP   0;
NETWORK
TITLE =

      A     M   1005.5;
      =     L      0.0;
      BLD   103;
      A     I    331.0;
      =     L      0.1;
      BLD   103;
      A     I    331.1;
      =     L      0.2;
      BLD   103;
      A     M   1243.2;
      =     L      2.1;
      BLD   103;
      A     M   1243.3;
      =     L      2.2;
      BLD   103;
      AN    M   1004.0;
      AN    M   1004.1;
      AN    M   6060.0;
      AN    M   6260.0;
      AN    M   6280.0;
      AN    M   1004.2;
      A     M   1000.2;
      =     L      2.3;
      BLD   103;
      A     I      0.1;
      =     L      2.5;
      BLD   103;
      A     M      0.5;
      =     L      2.6;
      BLD   103;
      CALL #S702_TL_DC_U262_1_UP_DN (
           Enable_Aux               := L      0.0,
           Adv_Amount               := 1,
           Ret_Amount               := 1,
           LS_Adv1                  := L      0.1,
           LS_Ret1                  := L      0.2,
           SOL_Adv                  := L      2.1,
           SOL_Ret                  := L      2.2,
           M_Ready                  := L      2.3,
           T_CHK1                   := T#4S,
           T_CHK2                   := T#4S,
           PB_Error_Rst             := L      2.5,
           M_FLICK                  := L      2.6,
           M_Adv_Err                := M   1253.2,
           M_Ret_Err                := M   1253.3,
           Visu_Adv                 := DB51.DBW  372,
           Visu_Ret                 := DB51.DBW  374);
      NOP   0;
NETWORK
TITLE =
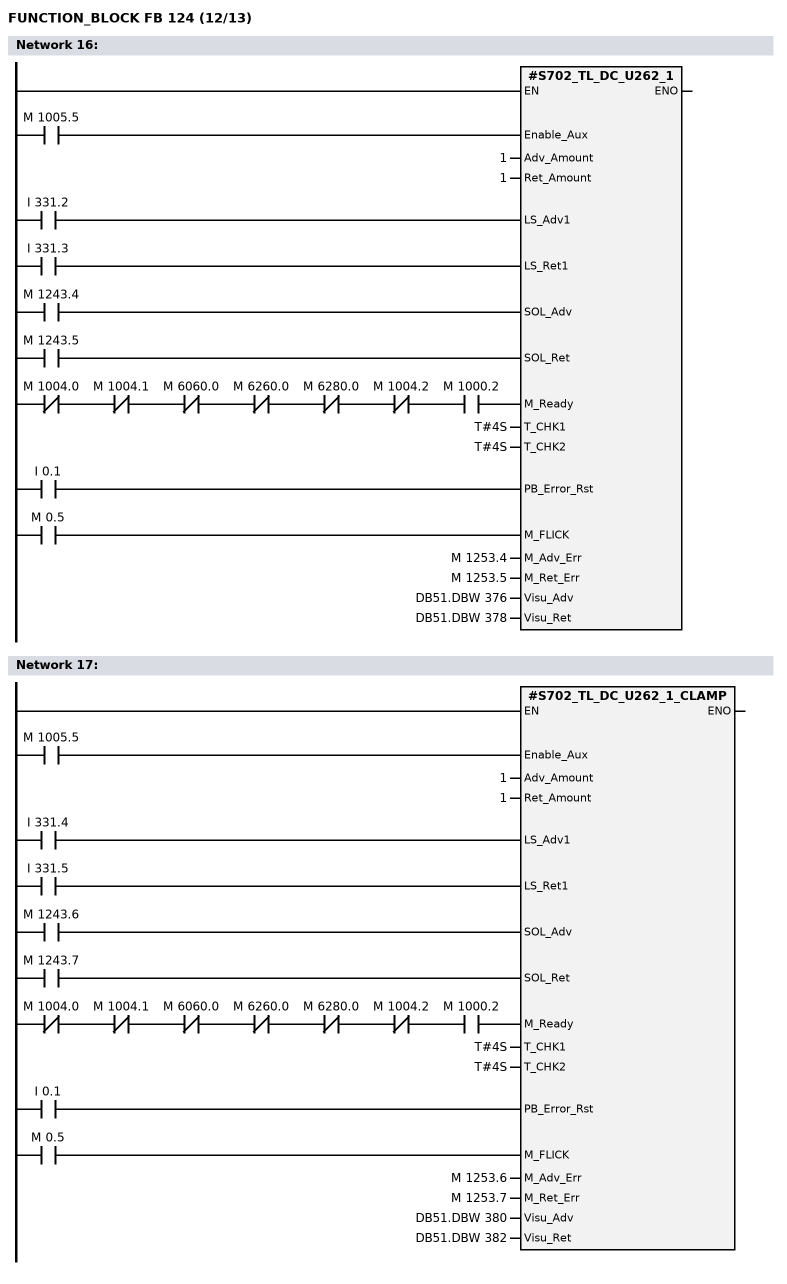

      A     M   1005.5;
      =     L      0.0;
      BLD   103;
      A     I    331.2;
      =     L      0.1;
      BLD   103;
      A     I    331.3;
      =     L      0.2;
      BLD   103;
      A     M   1243.4;
      =     L      2.1;
      BLD   103;
      A     M   1243.5;
      =     L      2.2;
      BLD   103;
      AN    M   1004.0;
      AN    M   1004.1;
      AN    M   6060.0;
      AN    M   6260.0;
      AN    M   6280.0;
      AN    M   1004.2;
      A     M   1000.2;
      =     L      2.3;
      BLD   103;
      A     I      0.1;
      =     L      2.5;
      BLD   103;
      A     M      0.5;
      =     L      2.6;
      BLD   103;
      CALL #S702_TL_DC_U262_1 (
           Enable_Aux               := L      0.0,
           Adv_Amount               := 1,
           Ret_Amount               := 1,
           LS_Adv1                  := L      0.1,
           LS_Ret1                  := L      0.2,
           SOL_Adv                  := L      2.1,
           SOL_Ret                  := L      2.2,
           M_Ready                  := L      2.3,
           T_CHK1                   := T#4S,
           T_CHK2                   := T#4S,
           PB_Error_Rst             := L      2.5,
           M_FLICK                  := L      2.6,
           M_Adv_Err                := M   1253.4,
           M_Ret_Err                := M   1253.5,
           Visu_Adv                 := DB51.DBW  376,
           Visu_Ret                 := DB51.DBW  378);
      NOP   0;
NETWORK
TITLE =

      A     M   1005.5;
      =     L      0.0;
      BLD   103;
      A     I    331.4;
      =     L      0.1;
      BLD   103;
      A     I    331.5;
      =     L      0.2;
      BLD   103;
      A     M   1243.6;
      =     L      2.1;
      BLD   103;
      A     M   1243.7;
      =     L      2.2;
      BLD   103;
      AN    M   1004.0;
      AN    M   1004.1;
      AN    M   6060.0;
      AN    M   6260.0;
      AN    M   6280.0;
      AN    M   1004.2;
      A     M   1000.2;
      =     L      2.3;
      BLD   103;
      A     I      0.1;
      =     L      2.5;
      BLD   103;
      A     M      0.5;
      =     L      2.6;
      BLD   103;
      CALL #S702_TL_DC_U262_1_CLAMP (
           Enable_Aux               := L      0.0,
           Adv_Amount               := 1,
           Ret_Amount               := 1,
           LS_Adv1                  := L      0.1,
           LS_Ret1                  := L      0.2,
           SOL_Adv                  := L      2.1,
           SOL_Ret                  := L      2.2,
           M_Ready                  := L      2.3,
           T_CHK1                   := T#4S,
           T_CHK2                   := T#4S,
           PB_Error_Rst             := L      2.5,
           M_FLICK                  := L      2.6,
           M_Adv_Err                := M   1253.6,
           M_Ret_Err                := M   1253.7,
           Visu_Adv                 := DB51.DBW  380,
           Visu_Ret                 := DB51.DBW  382);
      NOP   0;
NETWORK
TITLE =
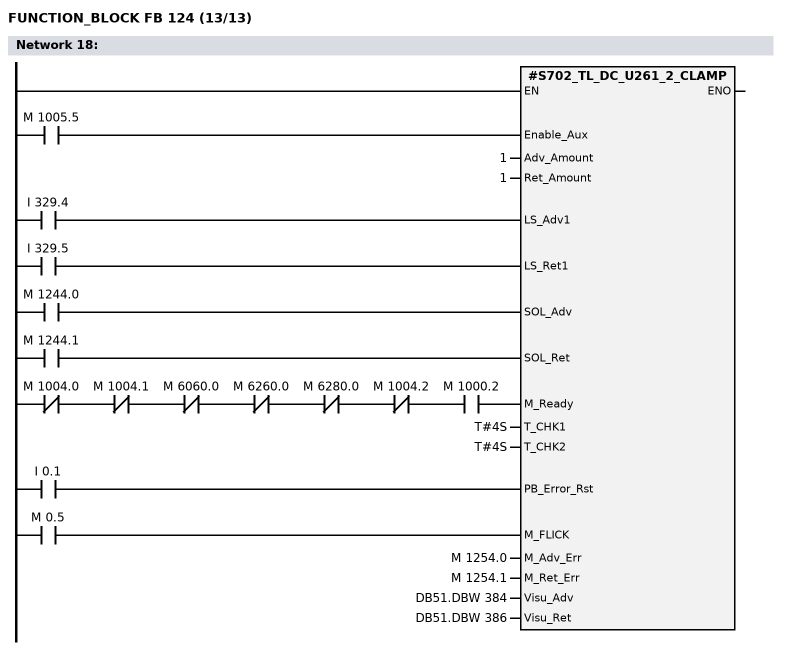

      A     M   1005.5;
      =     L      0.0;
      BLD   103;
      A     I    329.4;
      =     L      0.1;
      BLD   103;
      A     I    329.5;
      =     L      0.2;
      BLD   103;
      A     M   1244.0;
      =     L      2.1;
      BLD   103;
      A     M   1244.1;
      =     L      2.2;
      BLD   103;
      AN    M   1004.0;
      AN    M   1004.1;
      AN    M   6060.0;
      AN    M   6260.0;
      AN    M   6280.0;
      AN    M   1004.2;
      A     M   1000.2;
      =     L      2.3;
      BLD   103;
      A     I      0.1;
      =     L      2.5;
      BLD   103;
      A     M      0.5;
      =     L      2.6;
      BLD   103;
      CALL #S702_TL_DC_U261_2_CLAMP (
           Enable_Aux               := L      0.0,
           Adv_Amount               := 1,
           Ret_Amount               := 1,
           LS_Adv1                  := L      0.1,
           LS_Ret1                  := L      0.2,
           SOL_Adv                  := L      2.1,
           SOL_Ret                  := L      2.2,
           M_Ready                  := L      2.3,
           T_CHK1                   := T#4S,
           T_CHK2                   := T#4S,
           PB_Error_Rst             := L      2.5,
           M_FLICK                  := L      2.6,
           M_Adv_Err                := M   1254.0,
           M_Ret_Err                := M   1254.1,
           Visu_Adv                 := DB51.DBW  384,
           Visu_Ret                 := DB51.DBW  386);
      NOP   0;
END_FUNCTION_BLOCK

DATA_BLOCK DB 124
TITLE =
VERSION : 0.0

 FB 124
BEGIN
   S702_TL_DC_PIN.Enable_Aux := FALSE;
   S702_TL_DC_PIN.Adv_Amount := 0;
   S702_TL_DC_PIN.Ret_Amount := 0;
   S702_TL_DC_PIN.LS_Adv1 := FALSE;
   S702_TL_DC_PIN.LS_Ret1 := FALSE;
   S702_TL_DC_PIN.LS_Adv2 := FALSE;
   S702_TL_DC_PIN.LS_Ret2 := FALSE;
   S702_TL_DC_PIN.LS_Adv3 := FALSE;
   S702_TL_DC_PIN.LS_Ret3 := FALSE;
   S702_TL_DC_PIN.LS_Adv4 := FALSE;
   S702_TL_DC_PIN.LS_Ret4 := FALSE;
   S702_TL_DC_PIN.LS_Adv5 := FALSE;
   S702_TL_DC_PIN.LS_Ret5 := FALSE;
   S702_TL_DC_PIN.LS_Adv6 := FALSE;
   S702_TL_DC_PIN.LS_Ret6 := FALSE;
   S702_TL_DC_PIN.LS_Adv7 := FALSE;
   S702_TL_DC_PIN.LS_Ret7 := FALSE;
   S702_TL_DC_PIN.LS_Adv8 := FALSE;
   S702_TL_DC_PIN.LS_Ret8 := FALSE;
   S702_TL_DC_PIN.SOL_Adv := FALSE;
   S702_TL_DC_PIN.SOL_Ret := FALSE;
   S702_TL_DC_PIN.M_Ready := FALSE;
   S702_TL_DC_PIN.T_CHK1 := T#0MS;
   S702_TL_DC_PIN.T_CHK2 := T#0MS;
   S702_TL_DC_PIN.PB_Lamp_CHK := FALSE;
   S702_TL_DC_PIN.PB_Error_Rst := FALSE;
   S702_TL_DC_PIN.M_FLICK := FALSE;
   S702_TL_DC_PIN.M_Adv_Err := FALSE;
   S702_TL_DC_PIN.M_Ret_Err := FALSE;
   S702_TL_DC_PIN.LP_Adv := FALSE;
   S702_TL_DC_PIN.LP_Ret := FALSE;
   S702_TL_DC_PIN.Visu_Adv := W#16#0;
   S702_TL_DC_PIN.Visu_Ret := W#16#0;
   S702_TL_DC_PIN.Error_T1.IN := FALSE;
   S702_TL_DC_PIN.Error_T1.PT := T#0MS;
   S702_TL_DC_PIN.Error_T1.Q := FALSE;
   S702_TL_DC_PIN.Error_T1.ET := T#0MS;
   S702_TL_DC_PIN.Error_T1.STATE := B#16#0;
   S702_TL_DC_PIN.Error_T1.STIME := T#0MS;
   S702_TL_DC_PIN.Error_T1.ATIME := T#0MS;
   S702_TL_DC_PIN.Error_T2.IN := FALSE;
   S702_TL_DC_PIN.Error_T2.PT := T#0MS;
   S702_TL_DC_PIN.Error_T2.Q := FALSE;
   S702_TL_DC_PIN.Error_T2.ET := T#0MS;
   S702_TL_DC_PIN.Error_T2.STATE := B#16#0;
   S702_TL_DC_PIN.Error_T2.STIME := T#0MS;
   S702_TL_DC_PIN.Error_T2.ATIME := T#0MS;
   S702_TL_DC_PIN.Adv_End_Aux := FALSE;
   S702_TL_DC_PIN.Ret_End_Aux := FALSE;
   S702_TL_DC_PIN.CHK_Aux1 := FALSE;
   S702_TL_DC_PIN.CHK_Aux2 := FALSE;
   S702_TL_DC_PIN.Error_T1_DN := FALSE;
   S702_TL_DC_PIN.Error_T2_DN := FALSE;
   S702_TL_DC_PIN.Adv_Memo := FALSE;
   S702_TL_DC_PIN.Visu_Adv_Arr[0] := FALSE;
   S702_TL_DC_PIN.Visu_Adv_Arr[1] := FALSE;
   S702_TL_DC_PIN.Visu_Adv_Arr[2] := FALSE;
   S702_TL_DC_PIN.Visu_Adv_Arr[3] := FALSE;
   S702_TL_DC_PIN.Visu_Adv_Arr[4] := FALSE;
   S702_TL_DC_PIN.Visu_Adv_Arr[5] := FALSE;
   S702_TL_DC_PIN.Visu_Adv_Arr[6] := FALSE;
   S702_TL_DC_PIN.Visu_Adv_Arr[7] := FALSE;
   S702_TL_DC_PIN.Visu_Adv_Arr[8] := FALSE;
   S702_TL_DC_PIN.Visu_Adv_Arr[9] := FALSE;
   S702_TL_DC_PIN.Visu_Adv_Arr[10] := FALSE;
   S702_TL_DC_PIN.Visu_Adv_Arr[11] := FALSE;
   S702_TL_DC_PIN.Visu_Adv_Arr[12] := FALSE;
   S702_TL_DC_PIN.Visu_Adv_Arr[13] := FALSE;
   S702_TL_DC_PIN.Visu_Adv_Arr[14] := FALSE;
   S702_TL_DC_PIN.Visu_Adv_Arr[15] := FALSE;
   S702_TL_DC_PIN.Visu_Ret_Arr[0] := FALSE;
   S702_TL_DC_PIN.Visu_Ret_Arr[1] := FALSE;
   S702_TL_DC_PIN.Visu_Ret_Arr[2] := FALSE;
   S702_TL_DC_PIN.Visu_Ret_Arr[3] := FALSE;
   S702_TL_DC_PIN.Visu_Ret_Arr[4] := FALSE;
   S702_TL_DC_PIN.Visu_Ret_Arr[5] := FALSE;
   S702_TL_DC_PIN.Visu_Ret_Arr[6] := FALSE;
   S702_TL_DC_PIN.Visu_Ret_Arr[7] := FALSE;
   S702_TL_DC_PIN.Visu_Ret_Arr[8] := FALSE;
   S702_TL_DC_PIN.Visu_Ret_Arr[9] := FALSE;
   S702_TL_DC_PIN.Visu_Ret_Arr[10] := FALSE;
   S702_TL_DC_PIN.Visu_Ret_Arr[11] := FALSE;
   S702_TL_DC_PIN.Visu_Ret_Arr[12] := FALSE;
   S702_TL_DC_PIN.Visu_Ret_Arr[13] := FALSE;
   S702_TL_DC_PIN.Visu_Ret_Arr[14] := FALSE;
   S702_TL_DC_PIN.Visu_Ret_Arr[15] := FALSE;
   S702_TL_DC_PIN.BLK_Move_Ret := 0;
   S702_TL_DC_PIN.Enable := FALSE;
   S702_TL_DC_PIN.Adv_End := FALSE;
   S702_TL_DC_PIN.Ret_End := FALSE;
   S702_TL_DC_LATCH1.Enable_Aux := FALSE;
   S702_TL_DC_LATCH1.Adv_Amount := 0;
   S702_TL_DC_LATCH1.Ret_Amount := 0;
   S702_TL_DC_LATCH1.LS_Adv1 := FALSE;
   S702_TL_DC_LATCH1.LS_Ret1 := FALSE;
   S702_TL_DC_LATCH1.LS_Adv2 := FALSE;
   S702_TL_DC_LATCH1.LS_Ret2 := FALSE;
   S702_TL_DC_LATCH1.LS_Adv3 := FALSE;
   S702_TL_DC_LATCH1.LS_Ret3 := FALSE;
   S702_TL_DC_LATCH1.LS_Adv4 := FALSE;
   S702_TL_DC_LATCH1.LS_Ret4 := FALSE;
   S702_TL_DC_LATCH1.LS_Adv5 := FALSE;
   S702_TL_DC_LATCH1.LS_Ret5 := FALSE;
   S702_TL_DC_LATCH1.LS_Adv6 := FALSE;
   S702_TL_DC_LATCH1.LS_Ret6 := FALSE;
   S702_TL_DC_LATCH1.LS_Adv7 := FALSE;
   S702_TL_DC_LATCH1.LS_Ret7 := FALSE;
   S702_TL_DC_LATCH1.LS_Adv8 := FALSE;
   S702_TL_DC_LATCH1.LS_Ret8 := FALSE;
   S702_TL_DC_LATCH1.SOL_Adv := FALSE;
   S702_TL_DC_LATCH1.SOL_Ret := FALSE;
   S702_TL_DC_LATCH1.M_Ready := FALSE;
   S702_TL_DC_LATCH1.T_CHK1 := T#0MS;
   S702_TL_DC_LATCH1.T_CHK2 := T#0MS;
   S702_TL_DC_LATCH1.PB_Lamp_CHK := FALSE;
   S702_TL_DC_LATCH1.PB_Error_Rst := FALSE;
   S702_TL_DC_LATCH1.M_FLICK := FALSE;
   S702_TL_DC_LATCH1.M_Adv_Err := FALSE;
   S702_TL_DC_LATCH1.M_Ret_Err := FALSE;
   S702_TL_DC_LATCH1.LP_Adv := FALSE;
   S702_TL_DC_LATCH1.LP_Ret := FALSE;
   S702_TL_DC_LATCH1.Visu_Adv := W#16#0;
   S702_TL_DC_LATCH1.Visu_Ret := W#16#0;
   S702_TL_DC_LATCH1.Error_T1.IN := FALSE;
   S702_TL_DC_LATCH1.Error_T1.PT := T#0MS;
   S702_TL_DC_LATCH1.Error_T1.Q := FALSE;
   S702_TL_DC_LATCH1.Error_T1.ET := T#0MS;
   S702_TL_DC_LATCH1.Error_T1.STATE := B#16#0;
   S702_TL_DC_LATCH1.Error_T1.STIME := T#0MS;
   S702_TL_DC_LATCH1.Error_T1.ATIME := T#0MS;
   S702_TL_DC_LATCH1.Error_T2.IN := FALSE;
   S702_TL_DC_LATCH1.Error_T2.PT := T#0MS;
   S702_TL_DC_LATCH1.Error_T2.Q := FALSE;
   S702_TL_DC_LATCH1.Error_T2.ET := T#0MS;
   S702_TL_DC_LATCH1.Error_T2.STATE := B#16#0;
   S702_TL_DC_LATCH1.Error_T2.STIME := T#0MS;
   S702_TL_DC_LATCH1.Error_T2.ATIME := T#0MS;
   S702_TL_DC_LATCH1.Adv_End_Aux := FALSE;
   S702_TL_DC_LATCH1.Ret_End_Aux := FALSE;
   S702_TL_DC_LATCH1.CHK_Aux1 := FALSE;
   S702_TL_DC_LATCH1.CHK_Aux2 := FALSE;
   S702_TL_DC_LATCH1.Error_T1_DN := FALSE;
   S702_TL_DC_LATCH1.Error_T2_DN := FALSE;
   S702_TL_DC_LATCH1.Adv_Memo := FALSE;
   S702_TL_DC_LATCH1.Visu_Adv_Arr[0] := FALSE;
   S702_TL_DC_LATCH1.Visu_Adv_Arr[1] := FALSE;
   S702_TL_DC_LATCH1.Visu_Adv_Arr[2] := FALSE;
   S702_TL_DC_LATCH1.Visu_Adv_Arr[3] := FALSE;
   S702_TL_DC_LATCH1.Visu_Adv_Arr[4] := FALSE;
   S702_TL_DC_LATCH1.Visu_Adv_Arr[5] := FALSE;
   S702_TL_DC_LATCH1.Visu_Adv_Arr[6] := FALSE;
   S702_TL_DC_LATCH1.Visu_Adv_Arr[7] := FALSE;
   S702_TL_DC_LATCH1.Visu_Adv_Arr[8] := FALSE;
   S702_TL_DC_LATCH1.Visu_Adv_Arr[9] := FALSE;
   S702_TL_DC_LATCH1.Visu_Adv_Arr[10] := FALSE;
   S702_TL_DC_LATCH1.Visu_Adv_Arr[11] := FALSE;
   S702_TL_DC_LATCH1.Visu_Adv_Arr[12] := FALSE;
   S702_TL_DC_LATCH1.Visu_Adv_Arr[13] := FALSE;
   S702_TL_DC_LATCH1.Visu_Adv_Arr[14] := FALSE;
   S702_TL_DC_LATCH1.Visu_Adv_Arr[15] := FALSE;
   S702_TL_DC_LATCH1.Visu_Ret_Arr[0] := FALSE;
   S702_TL_DC_LATCH1.Visu_Ret_Arr[1] := FALSE;
   S702_TL_DC_LATCH1.Visu_Ret_Arr[2] := FALSE;
   S702_TL_DC_LATCH1.Visu_Ret_Arr[3] := FALSE;
   S702_TL_DC_LATCH1.Visu_Ret_Arr[4] := FALSE;
   S702_TL_DC_LATCH1.Visu_Ret_Arr[5] := FALSE;
   S702_TL_DC_LATCH1.Visu_Ret_Arr[6] := FALSE;
   S702_TL_DC_LATCH1.Visu_Ret_Arr[7] := FALSE;
   S702_TL_DC_LATCH1.Visu_Ret_Arr[8] := FALSE;
   S702_TL_DC_LATCH1.Visu_Ret_Arr[9] := FALSE;
   S702_TL_DC_LATCH1.Visu_Ret_Arr[10] := FALSE;
   S702_TL_DC_LATCH1.Visu_Ret_Arr[11] := FALSE;
   S702_TL_DC_LATCH1.Visu_Ret_Arr[12] := FALSE;
   S702_TL_DC_LATCH1.Visu_Ret_Arr[13] := FALSE;
   S702_TL_DC_LATCH1.Visu_Ret_Arr[14] := FALSE;
   S702_TL_DC_LATCH1.Visu_Ret_Arr[15] := FALSE;
   S702_TL_DC_LATCH1.BLK_Move_Ret := 0;
   S702_TL_DC_LATCH1.Enable := FALSE;
   S702_TL_DC_LATCH1.Adv_End := FALSE;
   S702_TL_DC_LATCH1.Ret_End := FALSE;
   S702_TL_DC_LATCH2.Enable_Aux := FALSE;
   S702_TL_DC_LATCH2.Adv_Amount := 0;
   S702_TL_DC_LATCH2.Ret_Amount := 0;
   S702_TL_DC_LATCH2.LS_Adv1 := FALSE;
   S702_TL_DC_LATCH2.LS_Ret1 := FALSE;
   S702_TL_DC_LATCH2.LS_Adv2 := FALSE;
   S702_TL_DC_LATCH2.LS_Ret2 := FALSE;
   S702_TL_DC_LATCH2.LS_Adv3 := FALSE;
   S702_TL_DC_LATCH2.LS_Ret3 := FALSE;
   S702_TL_DC_LATCH2.LS_Adv4 := FALSE;
   S702_TL_DC_LATCH2.LS_Ret4 := FALSE;
   S702_TL_DC_LATCH2.LS_Adv5 := FALSE;
   S702_TL_DC_LATCH2.LS_Ret5 := FALSE;
   S702_TL_DC_LATCH2.LS_Adv6 := FALSE;
   S702_TL_DC_LATCH2.LS_Ret6 := FALSE;
   S702_TL_DC_LATCH2.LS_Adv7 := FALSE;
   S702_TL_DC_LATCH2.LS_Ret7 := FALSE;
   S702_TL_DC_LATCH2.LS_Adv8 := FALSE;
   S702_TL_DC_LATCH2.LS_Ret8 := FALSE;
   S702_TL_DC_LATCH2.SOL_Adv := FALSE;
   S702_TL_DC_LATCH2.SOL_Ret := FALSE;
   S702_TL_DC_LATCH2.M_Ready := FALSE;
   S702_TL_DC_LATCH2.T_CHK1 := T#0MS;
   S702_TL_DC_LATCH2.T_CHK2 := T#0MS;
   S702_TL_DC_LATCH2.PB_Lamp_CHK := FALSE;
   S702_TL_DC_LATCH2.PB_Error_Rst := FALSE;
   S702_TL_DC_LATCH2.M_FLICK := FALSE;
   S702_TL_DC_LATCH2.M_Adv_Err := FALSE;
   S702_TL_DC_LATCH2.M_Ret_Err := FALSE;
   S702_TL_DC_LATCH2.LP_Adv := FALSE;
   S702_TL_DC_LATCH2.LP_Ret := FALSE;
   S702_TL_DC_LATCH2.Visu_Adv := W#16#0;
   S702_TL_DC_LATCH2.Visu_Ret := W#16#0;
   S702_TL_DC_LATCH2.Error_T1.IN := FALSE;
   S702_TL_DC_LATCH2.Error_T1.PT := T#0MS;
   S702_TL_DC_LATCH2.Error_T1.Q := FALSE;
   S702_TL_DC_LATCH2.Error_T1.ET := T#0MS;
   S702_TL_DC_LATCH2.Error_T1.STATE := B#16#0;
   S702_TL_DC_LATCH2.Error_T1.STIME := T#0MS;
   S702_TL_DC_LATCH2.Error_T1.ATIME := T#0MS;
   S702_TL_DC_LATCH2.Error_T2.IN := FALSE;
   S702_TL_DC_LATCH2.Error_T2.PT := T#0MS;
   S702_TL_DC_LATCH2.Error_T2.Q := FALSE;
   S702_TL_DC_LATCH2.Error_T2.ET := T#0MS;
   S702_TL_DC_LATCH2.Error_T2.STATE := B#16#0;
   S702_TL_DC_LATCH2.Error_T2.STIME := T#0MS;
   S702_TL_DC_LATCH2.Error_T2.ATIME := T#0MS;
   S702_TL_DC_LATCH2.Adv_End_Aux := FALSE;
   S702_TL_DC_LATCH2.Ret_End_Aux := FALSE;
   S702_TL_DC_LATCH2.CHK_Aux1 := FALSE;
   S702_TL_DC_LATCH2.CHK_Aux2 := FALSE;
   S702_TL_DC_LATCH2.Error_T1_DN := FALSE;
   S702_TL_DC_LATCH2.Error_T2_DN := FALSE;
   S702_TL_DC_LATCH2.Adv_Memo := FALSE;
   S702_TL_DC_LATCH2.Visu_Adv_Arr[0] := FALSE;
   S702_TL_DC_LATCH2.Visu_Adv_Arr[1] := FALSE;
   S702_TL_DC_LATCH2.Visu_Adv_Arr[2] := FALSE;
   S702_TL_DC_LATCH2.Visu_Adv_Arr[3] := FALSE;
   S702_TL_DC_LATCH2.Visu_Adv_Arr[4] := FALSE;
   S702_TL_DC_LATCH2.Visu_Adv_Arr[5] := FALSE;
   S702_TL_DC_LATCH2.Visu_Adv_Arr[6] := FALSE;
   S702_TL_DC_LATCH2.Visu_Adv_Arr[7] := FALSE;
   S702_TL_DC_LATCH2.Visu_Adv_Arr[8] := FALSE;
   S702_TL_DC_LATCH2.Visu_Adv_Arr[9] := FALSE;
   S702_TL_DC_LATCH2.Visu_Adv_Arr[10] := FALSE;
   S702_TL_DC_LATCH2.Visu_Adv_Arr[11] := FALSE;
   S702_TL_DC_LATCH2.Visu_Adv_Arr[12] := FALSE;
   S702_TL_DC_LATCH2.Visu_Adv_Arr[13] := FALSE;
   S702_TL_DC_LATCH2.Visu_Adv_Arr[14] := FALSE;
   S702_TL_DC_LATCH2.Visu_Adv_Arr[15] := FALSE;
   S702_TL_DC_LATCH2.Visu_Ret_Arr[0] := FALSE;
   S702_TL_DC_LATCH2.Visu_Ret_Arr[1] := FALSE;
   S702_TL_DC_LATCH2.Visu_Ret_Arr[2] := FALSE;
   S702_TL_DC_LATCH2.Visu_Ret_Arr[3] := FALSE;
   S702_TL_DC_LATCH2.Visu_Ret_Arr[4] := FALSE;
   S702_TL_DC_LATCH2.Visu_Ret_Arr[5] := FALSE;
   S702_TL_DC_LATCH2.Visu_Ret_Arr[6] := FALSE;
   S702_TL_DC_LATCH2.Visu_Ret_Arr[7] := FALSE;
   S702_TL_DC_LATCH2.Visu_Ret_Arr[8] := FALSE;
   S702_TL_DC_LATCH2.Visu_Ret_Arr[9] := FALSE;
   S702_TL_DC_LATCH2.Visu_Ret_Arr[10] := FALSE;
   S702_TL_DC_LATCH2.Visu_Ret_Arr[11] := FALSE;
   S702_TL_DC_LATCH2.Visu_Ret_Arr[12] := FALSE;
   S702_TL_DC_LATCH2.Visu_Ret_Arr[13] := FALSE;
   S702_TL_DC_LATCH2.Visu_Ret_Arr[14] := FALSE;
   S702_TL_DC_LATCH2.Visu_Ret_Arr[15] := FALSE;
   S702_TL_DC_LATCH2.BLK_Move_Ret := 0;
   S702_TL_DC_LATCH2.Enable := FALSE;
   S702_TL_DC_LATCH2.Adv_End := FALSE;
   S702_TL_DC_LATCH2.Ret_End := FALSE;
   S702_TL_DC_1ST_CLAMP1.Enable_Aux := FALSE;
   S702_TL_DC_1ST_CLAMP1.Adv_Amount := 0;
   S702_TL_DC_1ST_CLAMP1.Ret_Amount := 0;
   S702_TL_DC_1ST_CLAMP1.LS_Adv1 := FALSE;
   S702_TL_DC_1ST_CLAMP1.LS_Ret1 := FALSE;
   S702_TL_DC_1ST_CLAMP1.LS_Adv2 := FALSE;
   S702_TL_DC_1ST_CLAMP1.LS_Ret2 := FALSE;
   S702_TL_DC_1ST_CLAMP1.LS_Adv3 := FALSE;
   S702_TL_DC_1ST_CLAMP1.LS_Ret3 := FALSE;
   S702_TL_DC_1ST_CLAMP1.LS_Adv4 := FALSE;
   S702_TL_DC_1ST_CLAMP1.LS_Ret4 := FALSE;
   S702_TL_DC_1ST_CLAMP1.LS_Adv5 := FALSE;
   S702_TL_DC_1ST_CLAMP1.LS_Ret5 := FALSE;
   S702_TL_DC_1ST_CLAMP1.LS_Adv6 := FALSE;
   S702_TL_DC_1ST_CLAMP1.LS_Ret6 := FALSE;
   S702_TL_DC_1ST_CLAMP1.LS_Adv7 := FALSE;
   S702_TL_DC_1ST_CLAMP1.LS_Ret7 := FALSE;
   S702_TL_DC_1ST_CLAMP1.LS_Adv8 := FALSE;
   S702_TL_DC_1ST_CLAMP1.LS_Ret8 := FALSE;
   S702_TL_DC_1ST_CLAMP1.SOL_Adv := FALSE;
   S702_TL_DC_1ST_CLAMP1.SOL_Ret := FALSE;
   S702_TL_DC_1ST_CLAMP1.M_Ready := FALSE;
   S702_TL_DC_1ST_CLAMP1.T_CHK1 := T#0MS;
   S702_TL_DC_1ST_CLAMP1.T_CHK2 := T#0MS;
   S702_TL_DC_1ST_CLAMP1.PB_Lamp_CHK := FALSE;
   S702_TL_DC_1ST_CLAMP1.PB_Error_Rst := FALSE;
   S702_TL_DC_1ST_CLAMP1.M_FLICK := FALSE;
   S702_TL_DC_1ST_CLAMP1.M_Adv_Err := FALSE;
   S702_TL_DC_1ST_CLAMP1.M_Ret_Err := FALSE;
   S702_TL_DC_1ST_CLAMP1.LP_Adv := FALSE;
   S702_TL_DC_1ST_CLAMP1.LP_Ret := FALSE;
   S702_TL_DC_1ST_CLAMP1.Visu_Adv := W#16#0;
   S702_TL_DC_1ST_CLAMP1.Visu_Ret := W#16#0;
   S702_TL_DC_1ST_CLAMP1.Error_T1.IN := FALSE;
   S702_TL_DC_1ST_CLAMP1.Error_T1.PT := T#0MS;
   S702_TL_DC_1ST_CLAMP1.Error_T1.Q := FALSE;
   S702_TL_DC_1ST_CLAMP1.Error_T1.ET := T#0MS;
   S702_TL_DC_1ST_CLAMP1.Error_T1.STATE := B#16#0;
   S702_TL_DC_1ST_CLAMP1.Error_T1.STIME := T#0MS;
   S702_TL_DC_1ST_CLAMP1.Error_T1.ATIME := T#0MS;
   S702_TL_DC_1ST_CLAMP1.Error_T2.IN := FALSE;
   S702_TL_DC_1ST_CLAMP1.Error_T2.PT := T#0MS;
   S702_TL_DC_1ST_CLAMP1.Error_T2.Q := FALSE;
   S702_TL_DC_1ST_CLAMP1.Error_T2.ET := T#0MS;
   S702_TL_DC_1ST_CLAMP1.Error_T2.STATE := B#16#0;
   S702_TL_DC_1ST_CLAMP1.Error_T2.STIME := T#0MS;
   S702_TL_DC_1ST_CLAMP1.Error_T2.ATIME := T#0MS;
   S702_TL_DC_1ST_CLAMP1.Adv_End_Aux := FALSE;
   S702_TL_DC_1ST_CLAMP1.Ret_End_Aux := FALSE;
   S702_TL_DC_1ST_CLAMP1.CHK_Aux1 := FALSE;
   S702_TL_DC_1ST_CLAMP1.CHK_Aux2 := FALSE;
   S702_TL_DC_1ST_CLAMP1.Error_T1_DN := FALSE;
   S702_TL_DC_1ST_CLAMP1.Error_T2_DN := FALSE;
   S702_TL_DC_1ST_CLAMP1.Adv_Memo := FALSE;
   S702_TL_DC_1ST_CLAMP1.Visu_Adv_Arr[0] := FALSE;
   S702_TL_DC_1ST_CLAMP1.Visu_Adv_Arr[1] := FALSE;
   S702_TL_DC_1ST_CLAMP1.Visu_Adv_Arr[2] := FALSE;
   S702_TL_DC_1ST_CLAMP1.Visu_Adv_Arr[3] := FALSE;
   S702_TL_DC_1ST_CLAMP1.Visu_Adv_Arr[4] := FALSE;
   S702_TL_DC_1ST_CLAMP1.Visu_Adv_Arr[5] := FALSE;
   S702_TL_DC_1ST_CLAMP1.Visu_Adv_Arr[6] := FALSE;
   S702_TL_DC_1ST_CLAMP1.Visu_Adv_Arr[7] := FALSE;
   S702_TL_DC_1ST_CLAMP1.Visu_Adv_Arr[8] := FALSE;
   S702_TL_DC_1ST_CLAMP1.Visu_Adv_Arr[9] := FALSE;
   S702_TL_DC_1ST_CLAMP1.Visu_Adv_Arr[10] := FALSE;
   S702_TL_DC_1ST_CLAMP1.Visu_Adv_Arr[11] := FALSE;
   S702_TL_DC_1ST_CLAMP1.Visu_Adv_Arr[12] := FALSE;
   S702_TL_DC_1ST_CLAMP1.Visu_Adv_Arr[13] := FALSE;
   S702_TL_DC_1ST_CLAMP1.Visu_Adv_Arr[14] := FALSE;
   S702_TL_DC_1ST_CLAMP1.Visu_Adv_Arr[15] := FALSE;
   S702_TL_DC_1ST_CLAMP1.Visu_Ret_Arr[0] := FALSE;
   S702_TL_DC_1ST_CLAMP1.Visu_Ret_Arr[1] := FALSE;
   S702_TL_DC_1ST_CLAMP1.Visu_Ret_Arr[2] := FALSE;
   S702_TL_DC_1ST_CLAMP1.Visu_Ret_Arr[3] := FALSE;
   S702_TL_DC_1ST_CLAMP1.Visu_Ret_Arr[4] := FALSE;
   S702_TL_DC_1ST_CLAMP1.Visu_Ret_Arr[5] := FALSE;
   S702_TL_DC_1ST_CLAMP1.Visu_Ret_Arr[6] := FALSE;
   S702_TL_DC_1ST_CLAMP1.Visu_Ret_Arr[7] := FALSE;
   S702_TL_DC_1ST_CLAMP1.Visu_Ret_Arr[8] := FALSE;
   S702_TL_DC_1ST_CLAMP1.Visu_Ret_Arr[9] := FALSE;
   S702_TL_DC_1ST_CLAMP1.Visu_Ret_Arr[10] := FALSE;
   S702_TL_DC_1ST_CLAMP1.Visu_Ret_Arr[11] := FALSE;
   S702_TL_DC_1ST_CLAMP1.Visu_Ret_Arr[12] := FALSE;
   S702_TL_DC_1ST_CLAMP1.Visu_Ret_Arr[13] := FALSE;
   S702_TL_DC_1ST_CLAMP1.Visu_Ret_Arr[14] := FALSE;
   S702_TL_DC_1ST_CLAMP1.Visu_Ret_Arr[15] := FALSE;
   S702_TL_DC_1ST_CLAMP1.BLK_Move_Ret := 0;
   S702_TL_DC_1ST_CLAMP1.Enable := FALSE;
   S702_TL_DC_1ST_CLAMP1.Adv_End := FALSE;
   S702_TL_DC_1ST_CLAMP1.Ret_End := FALSE;
   S702_TL_DC_1ST_CLAMP2.Enable_Aux := FALSE;
   S702_TL_DC_1ST_CLAMP2.Adv_Amount := 0;
   S702_TL_DC_1ST_CLAMP2.Ret_Amount := 0;
   S702_TL_DC_1ST_CLAMP2.LS_Adv1 := FALSE;
   S702_TL_DC_1ST_CLAMP2.LS_Ret1 := FALSE;
   S702_TL_DC_1ST_CLAMP2.LS_Adv2 := FALSE;
   S702_TL_DC_1ST_CLAMP2.LS_Ret2 := FALSE;
   S702_TL_DC_1ST_CLAMP2.LS_Adv3 := FALSE;
   S702_TL_DC_1ST_CLAMP2.LS_Ret3 := FALSE;
   S702_TL_DC_1ST_CLAMP2.LS_Adv4 := FALSE;
   S702_TL_DC_1ST_CLAMP2.LS_Ret4 := FALSE;
   S702_TL_DC_1ST_CLAMP2.LS_Adv5 := FALSE;
   S702_TL_DC_1ST_CLAMP2.LS_Ret5 := FALSE;
   S702_TL_DC_1ST_CLAMP2.LS_Adv6 := FALSE;
   S702_TL_DC_1ST_CLAMP2.LS_Ret6 := FALSE;
   S702_TL_DC_1ST_CLAMP2.LS_Adv7 := FALSE;
   S702_TL_DC_1ST_CLAMP2.LS_Ret7 := FALSE;
   S702_TL_DC_1ST_CLAMP2.LS_Adv8 := FALSE;
   S702_TL_DC_1ST_CLAMP2.LS_Ret8 := FALSE;
   S702_TL_DC_1ST_CLAMP2.SOL_Adv := FALSE;
   S702_TL_DC_1ST_CLAMP2.SOL_Ret := FALSE;
   S702_TL_DC_1ST_CLAMP2.M_Ready := FALSE;
   S702_TL_DC_1ST_CLAMP2.T_CHK1 := T#0MS;
   S702_TL_DC_1ST_CLAMP2.T_CHK2 := T#0MS;
   S702_TL_DC_1ST_CLAMP2.PB_Lamp_CHK := FALSE;
   S702_TL_DC_1ST_CLAMP2.PB_Error_Rst := FALSE;
   S702_TL_DC_1ST_CLAMP2.M_FLICK := FALSE;
   S702_TL_DC_1ST_CLAMP2.M_Adv_Err := FALSE;
   S702_TL_DC_1ST_CLAMP2.M_Ret_Err := FALSE;
   S702_TL_DC_1ST_CLAMP2.LP_Adv := FALSE;
   S702_TL_DC_1ST_CLAMP2.LP_Ret := FALSE;
   S702_TL_DC_1ST_CLAMP2.Visu_Adv := W#16#0;
   S702_TL_DC_1ST_CLAMP2.Visu_Ret := W#16#0;
   S702_TL_DC_1ST_CLAMP2.Error_T1.IN := FALSE;
   S702_TL_DC_1ST_CLAMP2.Error_T1.PT := T#0MS;
   S702_TL_DC_1ST_CLAMP2.Error_T1.Q := FALSE;
   S702_TL_DC_1ST_CLAMP2.Error_T1.ET := T#0MS;
   S702_TL_DC_1ST_CLAMP2.Error_T1.STATE := B#16#0;
   S702_TL_DC_1ST_CLAMP2.Error_T1.STIME := T#0MS;
   S702_TL_DC_1ST_CLAMP2.Error_T1.ATIME := T#0MS;
   S702_TL_DC_1ST_CLAMP2.Error_T2.IN := FALSE;
   S702_TL_DC_1ST_CLAMP2.Error_T2.PT := T#0MS;
   S702_TL_DC_1ST_CLAMP2.Error_T2.Q := FALSE;
   S702_TL_DC_1ST_CLAMP2.Error_T2.ET := T#0MS;
   S702_TL_DC_1ST_CLAMP2.Error_T2.STATE := B#16#0;
   S702_TL_DC_1ST_CLAMP2.Error_T2.STIME := T#0MS;
   S702_TL_DC_1ST_CLAMP2.Error_T2.ATIME := T#0MS;
   S702_TL_DC_1ST_CLAMP2.Adv_End_Aux := FALSE;
   S702_TL_DC_1ST_CLAMP2.Ret_End_Aux := FALSE;
   S702_TL_DC_1ST_CLAMP2.CHK_Aux1 := FALSE;
   S702_TL_DC_1ST_CLAMP2.CHK_Aux2 := FALSE;
   S702_TL_DC_1ST_CLAMP2.Error_T1_DN := FALSE;
   S702_TL_DC_1ST_CLAMP2.Error_T2_DN := FALSE;
   S702_TL_DC_1ST_CLAMP2.Adv_Memo := FALSE;
   S702_TL_DC_1ST_CLAMP2.Visu_Adv_Arr[0] := FALSE;
   S702_TL_DC_1ST_CLAMP2.Visu_Adv_Arr[1] := FALSE;
   S702_TL_DC_1ST_CLAMP2.Visu_Adv_Arr[2] := FALSE;
   S702_TL_DC_1ST_CLAMP2.Visu_Adv_Arr[3] := FALSE;
   S702_TL_DC_1ST_CLAMP2.Visu_Adv_Arr[4] := FALSE;
   S702_TL_DC_1ST_CLAMP2.Visu_Adv_Arr[5] := FALSE;
   S702_TL_DC_1ST_CLAMP2.Visu_Adv_Arr[6] := FALSE;
   S702_TL_DC_1ST_CLAMP2.Visu_Adv_Arr[7] := FALSE;
   S702_TL_DC_1ST_CLAMP2.Visu_Adv_Arr[8] := FALSE;
   S702_TL_DC_1ST_CLAMP2.Visu_Adv_Arr[9] := FALSE;
   S702_TL_DC_1ST_CLAMP2.Visu_Adv_Arr[10] := FALSE;
   S702_TL_DC_1ST_CLAMP2.Visu_Adv_Arr[11] := FALSE;
   S702_TL_DC_1ST_CLAMP2.Visu_Adv_Arr[12] := FALSE;
   S702_TL_DC_1ST_CLAMP2.Visu_Adv_Arr[13] := FALSE;
   S702_TL_DC_1ST_CLAMP2.Visu_Adv_Arr[14] := FALSE;
   S702_TL_DC_1ST_CLAMP2.Visu_Adv_Arr[15] := FALSE;
   S702_TL_DC_1ST_CLAMP2.Visu_Ret_Arr[0] := FALSE;
   S702_TL_DC_1ST_CLAMP2.Visu_Ret_Arr[1] := FALSE;
   S702_TL_DC_1ST_CLAMP2.Visu_Ret_Arr[2] := FALSE;
   S702_TL_DC_1ST_CLAMP2.Visu_Ret_Arr[3] := FALSE;
   S702_TL_DC_1ST_CLAMP2.Visu_Ret_Arr[4] := FALSE;
   S702_TL_DC_1ST_CLAMP2.Visu_Ret_Arr[5] := FALSE;
   S702_TL_DC_1ST_CLAMP2.Visu_Ret_Arr[6] := FALSE;
   S702_TL_DC_1ST_CLAMP2.Visu_Ret_Arr[7] := FALSE;
   S702_TL_DC_1ST_CLAMP2.Visu_Ret_Arr[8] := FALSE;
   S702_TL_DC_1ST_CLAMP2.Visu_Ret_Arr[9] := FALSE;
   S702_TL_DC_1ST_CLAMP2.Visu_Ret_Arr[10] := FALSE;
   S702_TL_DC_1ST_CLAMP2.Visu_Ret_Arr[11] := FALSE;
   S702_TL_DC_1ST_CLAMP2.Visu_Ret_Arr[12] := FALSE;
   S702_TL_DC_1ST_CLAMP2.Visu_Ret_Arr[13] := FALSE;
   S702_TL_DC_1ST_CLAMP2.Visu_Ret_Arr[14] := FALSE;
   S702_TL_DC_1ST_CLAMP2.Visu_Ret_Arr[15] := FALSE;
   S702_TL_DC_1ST_CLAMP2.BLK_Move_Ret := 0;
   S702_TL_DC_1ST_CLAMP2.Enable := FALSE;
   S702_TL_DC_1ST_CLAMP2.Adv_End := FALSE;
   S702_TL_DC_1ST_CLAMP2.Ret_End := FALSE;
   S702_TL_DC_1ST_CLAMP3.Enable_Aux := FALSE;
   S702_TL_DC_1ST_CLAMP3.Adv_Amount := 0;
   S702_TL_DC_1ST_CLAMP3.Ret_Amount := 0;
   S702_TL_DC_1ST_CLAMP3.LS_Adv1 := FALSE;
   S702_TL_DC_1ST_CLAMP3.LS_Ret1 := FALSE;
   S702_TL_DC_1ST_CLAMP3.LS_Adv2 := FALSE;
   S702_TL_DC_1ST_CLAMP3.LS_Ret2 := FALSE;
   S702_TL_DC_1ST_CLAMP3.LS_Adv3 := FALSE;
   S702_TL_DC_1ST_CLAMP3.LS_Ret3 := FALSE;
   S702_TL_DC_1ST_CLAMP3.LS_Adv4 := FALSE;
   S702_TL_DC_1ST_CLAMP3.LS_Ret4 := FALSE;
   S702_TL_DC_1ST_CLAMP3.LS_Adv5 := FALSE;
   S702_TL_DC_1ST_CLAMP3.LS_Ret5 := FALSE;
   S702_TL_DC_1ST_CLAMP3.LS_Adv6 := FALSE;
   S702_TL_DC_1ST_CLAMP3.LS_Ret6 := FALSE;
   S702_TL_DC_1ST_CLAMP3.LS_Adv7 := FALSE;
   S702_TL_DC_1ST_CLAMP3.LS_Ret7 := FALSE;
   S702_TL_DC_1ST_CLAMP3.LS_Adv8 := FALSE;
   S702_TL_DC_1ST_CLAMP3.LS_Ret8 := FALSE;
   S702_TL_DC_1ST_CLAMP3.SOL_Adv := FALSE;
   S702_TL_DC_1ST_CLAMP3.SOL_Ret := FALSE;
   S702_TL_DC_1ST_CLAMP3.M_Ready := FALSE;
   S702_TL_DC_1ST_CLAMP3.T_CHK1 := T#0MS;
   S702_TL_DC_1ST_CLAMP3.T_CHK2 := T#0MS;
   S702_TL_DC_1ST_CLAMP3.PB_Lamp_CHK := FALSE;
   S702_TL_DC_1ST_CLAMP3.PB_Error_Rst := FALSE;
   S702_TL_DC_1ST_CLAMP3.M_FLICK := FALSE;
   S702_TL_DC_1ST_CLAMP3.M_Adv_Err := FALSE;
   S702_TL_DC_1ST_CLAMP3.M_Ret_Err := FALSE;
   S702_TL_DC_1ST_CLAMP3.LP_Adv := FALSE;
   S702_TL_DC_1ST_CLAMP3.LP_Ret := FALSE;
   S702_TL_DC_1ST_CLAMP3.Visu_Adv := W#16#0;
   S702_TL_DC_1ST_CLAMP3.Visu_Ret := W#16#0;
   S702_TL_DC_1ST_CLAMP3.Error_T1.IN := FALSE;
   S702_TL_DC_1ST_CLAMP3.Error_T1.PT := T#0MS;
   S702_TL_DC_1ST_CLAMP3.Error_T1.Q := FALSE;
   S702_TL_DC_1ST_CLAMP3.Error_T1.ET := T#0MS;
   S702_TL_DC_1ST_CLAMP3.Error_T1.STATE := B#16#0;
   S702_TL_DC_1ST_CLAMP3.Error_T1.STIME := T#0MS;
   S702_TL_DC_1ST_CLAMP3.Error_T1.ATIME := T#0MS;
   S702_TL_DC_1ST_CLAMP3.Error_T2.IN := FALSE;
   S702_TL_DC_1ST_CLAMP3.Error_T2.PT := T#0MS;
   S702_TL_DC_1ST_CLAMP3.Error_T2.Q := FALSE;
   S702_TL_DC_1ST_CLAMP3.Error_T2.ET := T#0MS;
   S702_TL_DC_1ST_CLAMP3.Error_T2.STATE := B#16#0;
   S702_TL_DC_1ST_CLAMP3.Error_T2.STIME := T#0MS;
   S702_TL_DC_1ST_CLAMP3.Error_T2.ATIME := T#0MS;
   S702_TL_DC_1ST_CLAMP3.Adv_End_Aux := FALSE;
   S702_TL_DC_1ST_CLAMP3.Ret_End_Aux := FALSE;
   S702_TL_DC_1ST_CLAMP3.CHK_Aux1 := FALSE;
   S702_TL_DC_1ST_CLAMP3.CHK_Aux2 := FALSE;
   S702_TL_DC_1ST_CLAMP3.Error_T1_DN := FALSE;
   S702_TL_DC_1ST_CLAMP3.Error_T2_DN := FALSE;
   S702_TL_DC_1ST_CLAMP3.Adv_Memo := FALSE;
   S702_TL_DC_1ST_CLAMP3.Visu_Adv_Arr[0] := FALSE;
   S702_TL_DC_1ST_CLAMP3.Visu_Adv_Arr[1] := FALSE;
   S702_TL_DC_1ST_CLAMP3.Visu_Adv_Arr[2] := FALSE;
   S702_TL_DC_1ST_CLAMP3.Visu_Adv_Arr[3] := FALSE;
   S702_TL_DC_1ST_CLAMP3.Visu_Adv_Arr[4] := FALSE;
   S702_TL_DC_1ST_CLAMP3.Visu_Adv_Arr[5] := FALSE;
   S702_TL_DC_1ST_CLAMP3.Visu_Adv_Arr[6] := FALSE;
   S702_TL_DC_1ST_CLAMP3.Visu_Adv_Arr[7] := FALSE;
   S702_TL_DC_1ST_CLAMP3.Visu_Adv_Arr[8] := FALSE;
   S702_TL_DC_1ST_CLAMP3.Visu_Adv_Arr[9] := FALSE;
   S702_TL_DC_1ST_CLAMP3.Visu_Adv_Arr[10] := FALSE;
   S702_TL_DC_1ST_CLAMP3.Visu_Adv_Arr[11] := FALSE;
   S702_TL_DC_1ST_CLAMP3.Visu_Adv_Arr[12] := FALSE;
   S702_TL_DC_1ST_CLAMP3.Visu_Adv_Arr[13] := FALSE;
   S702_TL_DC_1ST_CLAMP3.Visu_Adv_Arr[14] := FALSE;
   S702_TL_DC_1ST_CLAMP3.Visu_Adv_Arr[15] := FALSE;
   S702_TL_DC_1ST_CLAMP3.Visu_Ret_Arr[0] := FALSE;
   S702_TL_DC_1ST_CLAMP3.Visu_Ret_Arr[1] := FALSE;
   S702_TL_DC_1ST_CLAMP3.Visu_Ret_Arr[2] := FALSE;
   S702_TL_DC_1ST_CLAMP3.Visu_Ret_Arr[3] := FALSE;
   S702_TL_DC_1ST_CLAMP3.Visu_Ret_Arr[4] := FALSE;
   S702_TL_DC_1ST_CLAMP3.Visu_Ret_Arr[5] := FALSE;
   S702_TL_DC_1ST_CLAMP3.Visu_Ret_Arr[6] := FALSE;
   S702_TL_DC_1ST_CLAMP3.Visu_Ret_Arr[7] := FALSE;
   S702_TL_DC_1ST_CLAMP3.Visu_Ret_Arr[8] := FALSE;
   S702_TL_DC_1ST_CLAMP3.Visu_Ret_Arr[9] := FALSE;
   S702_TL_DC_1ST_CLAMP3.Visu_Ret_Arr[10] := FALSE;
   S702_TL_DC_1ST_CLAMP3.Visu_Ret_Arr[11] := FALSE;
   S702_TL_DC_1ST_CLAMP3.Visu_Ret_Arr[12] := FALSE;
   S702_TL_DC_1ST_CLAMP3.Visu_Ret_Arr[13] := FALSE;
   S702_TL_DC_1ST_CLAMP3.Visu_Ret_Arr[14] := FALSE;
   S702_TL_DC_1ST_CLAMP3.Visu_Ret_Arr[15] := FALSE;
   S702_TL_DC_1ST_CLAMP3.BLK_Move_Ret := 0;
   S702_TL_DC_1ST_CLAMP3.Enable := FALSE;
   S702_TL_DC_1ST_CLAMP3.Adv_End := FALSE;
   S702_TL_DC_1ST_CLAMP3.Ret_End := FALSE;
   S702_TL_DC_2ND_CLAMP1.Enable_Aux := FALSE;
   S702_TL_DC_2ND_CLAMP1.Adv_Amount := 0;
   S702_TL_DC_2ND_CLAMP1.Ret_Amount := 0;
   S702_TL_DC_2ND_CLAMP1.LS_Adv1 := FALSE;
   S702_TL_DC_2ND_CLAMP1.LS_Ret1 := FALSE;
   S702_TL_DC_2ND_CLAMP1.LS_Adv2 := FALSE;
   S702_TL_DC_2ND_CLAMP1.LS_Ret2 := FALSE;
   S702_TL_DC_2ND_CLAMP1.LS_Adv3 := FALSE;
   S702_TL_DC_2ND_CLAMP1.LS_Ret3 := FALSE;
   S702_TL_DC_2ND_CLAMP1.LS_Adv4 := FALSE;
   S702_TL_DC_2ND_CLAMP1.LS_Ret4 := FALSE;
   S702_TL_DC_2ND_CLAMP1.LS_Adv5 := FALSE;
   S702_TL_DC_2ND_CLAMP1.LS_Ret5 := FALSE;
   S702_TL_DC_2ND_CLAMP1.LS_Adv6 := FALSE;
   S702_TL_DC_2ND_CLAMP1.LS_Ret6 := FALSE;
   S702_TL_DC_2ND_CLAMP1.LS_Adv7 := FALSE;
   S702_TL_DC_2ND_CLAMP1.LS_Ret7 := FALSE;
   S702_TL_DC_2ND_CLAMP1.LS_Adv8 := FALSE;
   S702_TL_DC_2ND_CLAMP1.LS_Ret8 := FALSE;
   S702_TL_DC_2ND_CLAMP1.SOL_Adv := FALSE;
   S702_TL_DC_2ND_CLAMP1.SOL_Ret := FALSE;
   S702_TL_DC_2ND_CLAMP1.M_Ready := FALSE;
   S702_TL_DC_2ND_CLAMP1.T_CHK1 := T#0MS;
   S702_TL_DC_2ND_CLAMP1.T_CHK2 := T#0MS;
   S702_TL_DC_2ND_CLAMP1.PB_Lamp_CHK := FALSE;
   S702_TL_DC_2ND_CLAMP1.PB_Error_Rst := FALSE;
   S702_TL_DC_2ND_CLAMP1.M_FLICK := FALSE;
   S702_TL_DC_2ND_CLAMP1.M_Adv_Err := FALSE;
   S702_TL_DC_2ND_CLAMP1.M_Ret_Err := FALSE;
   S702_TL_DC_2ND_CLAMP1.LP_Adv := FALSE;
   S702_TL_DC_2ND_CLAMP1.LP_Ret := FALSE;
   S702_TL_DC_2ND_CLAMP1.Visu_Adv := W#16#0;
   S702_TL_DC_2ND_CLAMP1.Visu_Ret := W#16#0;
   S702_TL_DC_2ND_CLAMP1.Error_T1.IN := FALSE;
   S702_TL_DC_2ND_CLAMP1.Error_T1.PT := T#0MS;
   S702_TL_DC_2ND_CLAMP1.Error_T1.Q := FALSE;
   S702_TL_DC_2ND_CLAMP1.Error_T1.ET := T#0MS;
   S702_TL_DC_2ND_CLAMP1.Error_T1.STATE := B#16#0;
   S702_TL_DC_2ND_CLAMP1.Error_T1.STIME := T#0MS;
   S702_TL_DC_2ND_CLAMP1.Error_T1.ATIME := T#0MS;
   S702_TL_DC_2ND_CLAMP1.Error_T2.IN := FALSE;
   S702_TL_DC_2ND_CLAMP1.Error_T2.PT := T#0MS;
   S702_TL_DC_2ND_CLAMP1.Error_T2.Q := FALSE;
   S702_TL_DC_2ND_CLAMP1.Error_T2.ET := T#0MS;
   S702_TL_DC_2ND_CLAMP1.Error_T2.STATE := B#16#0;
   S702_TL_DC_2ND_CLAMP1.Error_T2.STIME := T#0MS;
   S702_TL_DC_2ND_CLAMP1.Error_T2.ATIME := T#0MS;
   S702_TL_DC_2ND_CLAMP1.Adv_End_Aux := FALSE;
   S702_TL_DC_2ND_CLAMP1.Ret_End_Aux := FALSE;
   S702_TL_DC_2ND_CLAMP1.CHK_Aux1 := FALSE;
   S702_TL_DC_2ND_CLAMP1.CHK_Aux2 := FALSE;
   S702_TL_DC_2ND_CLAMP1.Error_T1_DN := FALSE;
   S702_TL_DC_2ND_CLAMP1.Error_T2_DN := FALSE;
   S702_TL_DC_2ND_CLAMP1.Adv_Memo := FALSE;
   S702_TL_DC_2ND_CLAMP1.Visu_Adv_Arr[0] := FALSE;
   S702_TL_DC_2ND_CLAMP1.Visu_Adv_Arr[1] := FALSE;
   S702_TL_DC_2ND_CLAMP1.Visu_Adv_Arr[2] := FALSE;
   S702_TL_DC_2ND_CLAMP1.Visu_Adv_Arr[3] := FALSE;
   S702_TL_DC_2ND_CLAMP1.Visu_Adv_Arr[4] := FALSE;
   S702_TL_DC_2ND_CLAMP1.Visu_Adv_Arr[5] := FALSE;
   S702_TL_DC_2ND_CLAMP1.Visu_Adv_Arr[6] := FALSE;
   S702_TL_DC_2ND_CLAMP1.Visu_Adv_Arr[7] := FALSE;
   S702_TL_DC_2ND_CLAMP1.Visu_Adv_Arr[8] := FALSE;
   S702_TL_DC_2ND_CLAMP1.Visu_Adv_Arr[9] := FALSE;
   S702_TL_DC_2ND_CLAMP1.Visu_Adv_Arr[10] := FALSE;
   S702_TL_DC_2ND_CLAMP1.Visu_Adv_Arr[11] := FALSE;
   S702_TL_DC_2ND_CLAMP1.Visu_Adv_Arr[12] := FALSE;
   S702_TL_DC_2ND_CLAMP1.Visu_Adv_Arr[13] := FALSE;
   S702_TL_DC_2ND_CLAMP1.Visu_Adv_Arr[14] := FALSE;
   S702_TL_DC_2ND_CLAMP1.Visu_Adv_Arr[15] := FALSE;
   S702_TL_DC_2ND_CLAMP1.Visu_Ret_Arr[0] := FALSE;
   S702_TL_DC_2ND_CLAMP1.Visu_Ret_Arr[1] := FALSE;
   S702_TL_DC_2ND_CLAMP1.Visu_Ret_Arr[2] := FALSE;
   S702_TL_DC_2ND_CLAMP1.Visu_Ret_Arr[3] := FALSE;
   S702_TL_DC_2ND_CLAMP1.Visu_Ret_Arr[4] := FALSE;
   S702_TL_DC_2ND_CLAMP1.Visu_Ret_Arr[5] := FALSE;
   S702_TL_DC_2ND_CLAMP1.Visu_Ret_Arr[6] := FALSE;
   S702_TL_DC_2ND_CLAMP1.Visu_Ret_Arr[7] := FALSE;
   S702_TL_DC_2ND_CLAMP1.Visu_Ret_Arr[8] := FALSE;
   S702_TL_DC_2ND_CLAMP1.Visu_Ret_Arr[9] := FALSE;
   S702_TL_DC_2ND_CLAMP1.Visu_Ret_Arr[10] := FALSE;
   S702_TL_DC_2ND_CLAMP1.Visu_Ret_Arr[11] := FALSE;
   S702_TL_DC_2ND_CLAMP1.Visu_Ret_Arr[12] := FALSE;
   S702_TL_DC_2ND_CLAMP1.Visu_Ret_Arr[13] := FALSE;
   S702_TL_DC_2ND_CLAMP1.Visu_Ret_Arr[14] := FALSE;
   S702_TL_DC_2ND_CLAMP1.Visu_Ret_Arr[15] := FALSE;
   S702_TL_DC_2ND_CLAMP1.BLK_Move_Ret := 0;
   S702_TL_DC_2ND_CLAMP1.Enable := FALSE;
   S702_TL_DC_2ND_CLAMP1.Adv_End := FALSE;
   S702_TL_DC_2ND_CLAMP1.Ret_End := FALSE;
   S702_TL_DC_2ND_CLAMP2.Enable_Aux := FALSE;
   S702_TL_DC_2ND_CLAMP2.Adv_Amount := 0;
   S702_TL_DC_2ND_CLAMP2.Ret_Amount := 0;
   S702_TL_DC_2ND_CLAMP2.LS_Adv1 := FALSE;
   S702_TL_DC_2ND_CLAMP2.LS_Ret1 := FALSE;
   S702_TL_DC_2ND_CLAMP2.LS_Adv2 := FALSE;
   S702_TL_DC_2ND_CLAMP2.LS_Ret2 := FALSE;
   S702_TL_DC_2ND_CLAMP2.LS_Adv3 := FALSE;
   S702_TL_DC_2ND_CLAMP2.LS_Ret3 := FALSE;
   S702_TL_DC_2ND_CLAMP2.LS_Adv4 := FALSE;
   S702_TL_DC_2ND_CLAMP2.LS_Ret4 := FALSE;
   S702_TL_DC_2ND_CLAMP2.LS_Adv5 := FALSE;
   S702_TL_DC_2ND_CLAMP2.LS_Ret5 := FALSE;
   S702_TL_DC_2ND_CLAMP2.LS_Adv6 := FALSE;
   S702_TL_DC_2ND_CLAMP2.LS_Ret6 := FALSE;
   S702_TL_DC_2ND_CLAMP2.LS_Adv7 := FALSE;
   S702_TL_DC_2ND_CLAMP2.LS_Ret7 := FALSE;
   S702_TL_DC_2ND_CLAMP2.LS_Adv8 := FALSE;
   S702_TL_DC_2ND_CLAMP2.LS_Ret8 := FALSE;
   S702_TL_DC_2ND_CLAMP2.SOL_Adv := FALSE;
   S702_TL_DC_2ND_CLAMP2.SOL_Ret := FALSE;
   S702_TL_DC_2ND_CLAMP2.M_Ready := FALSE;
   S702_TL_DC_2ND_CLAMP2.T_CHK1 := T#0MS;
   S702_TL_DC_2ND_CLAMP2.T_CHK2 := T#0MS;
   S702_TL_DC_2ND_CLAMP2.PB_Lamp_CHK := FALSE;
   S702_TL_DC_2ND_CLAMP2.PB_Error_Rst := FALSE;
   S702_TL_DC_2ND_CLAMP2.M_FLICK := FALSE;
   S702_TL_DC_2ND_CLAMP2.M_Adv_Err := FALSE;
   S702_TL_DC_2ND_CLAMP2.M_Ret_Err := FALSE;
   S702_TL_DC_2ND_CLAMP2.LP_Adv := FALSE;
   S702_TL_DC_2ND_CLAMP2.LP_Ret := FALSE;
   S702_TL_DC_2ND_CLAMP2.Visu_Adv := W#16#0;
   S702_TL_DC_2ND_CLAMP2.Visu_Ret := W#16#0;
   S702_TL_DC_2ND_CLAMP2.Error_T1.IN := FALSE;
   S702_TL_DC_2ND_CLAMP2.Error_T1.PT := T#0MS;
   S702_TL_DC_2ND_CLAMP2.Error_T1.Q := FALSE;
   S702_TL_DC_2ND_CLAMP2.Error_T1.ET := T#0MS;
   S702_TL_DC_2ND_CLAMP2.Error_T1.STATE := B#16#0;
   S702_TL_DC_2ND_CLAMP2.Error_T1.STIME := T#0MS;
   S702_TL_DC_2ND_CLAMP2.Error_T1.ATIME := T#0MS;
   S702_TL_DC_2ND_CLAMP2.Error_T2.IN := FALSE;
   S702_TL_DC_2ND_CLAMP2.Error_T2.PT := T#0MS;
   S702_TL_DC_2ND_CLAMP2.Error_T2.Q := FALSE;
   S702_TL_DC_2ND_CLAMP2.Error_T2.ET := T#0MS;
   S702_TL_DC_2ND_CLAMP2.Error_T2.STATE := B#16#0;
   S702_TL_DC_2ND_CLAMP2.Error_T2.STIME := T#0MS;
   S702_TL_DC_2ND_CLAMP2.Error_T2.ATIME := T#0MS;
   S702_TL_DC_2ND_CLAMP2.Adv_End_Aux := FALSE;
   S702_TL_DC_2ND_CLAMP2.Ret_End_Aux := FALSE;
   S702_TL_DC_2ND_CLAMP2.CHK_Aux1 := FALSE;
   S702_TL_DC_2ND_CLAMP2.CHK_Aux2 := FALSE;
   S702_TL_DC_2ND_CLAMP2.Error_T1_DN := FALSE;
   S702_TL_DC_2ND_CLAMP2.Error_T2_DN := FALSE;
   S702_TL_DC_2ND_CLAMP2.Adv_Memo := FALSE;
   S702_TL_DC_2ND_CLAMP2.Visu_Adv_Arr[0] := FALSE;
   S702_TL_DC_2ND_CLAMP2.Visu_Adv_Arr[1] := FALSE;
   S702_TL_DC_2ND_CLAMP2.Visu_Adv_Arr[2] := FALSE;
   S702_TL_DC_2ND_CLAMP2.Visu_Adv_Arr[3] := FALSE;
   S702_TL_DC_2ND_CLAMP2.Visu_Adv_Arr[4] := FALSE;
   S702_TL_DC_2ND_CLAMP2.Visu_Adv_Arr[5] := FALSE;
   S702_TL_DC_2ND_CLAMP2.Visu_Adv_Arr[6] := FALSE;
   S702_TL_DC_2ND_CLAMP2.Visu_Adv_Arr[7] := FALSE;
   S702_TL_DC_2ND_CLAMP2.Visu_Adv_Arr[8] := FALSE;
   S702_TL_DC_2ND_CLAMP2.Visu_Adv_Arr[9] := FALSE;
   S702_TL_DC_2ND_CLAMP2.Visu_Adv_Arr[10] := FALSE;
   S702_TL_DC_2ND_CLAMP2.Visu_Adv_Arr[11] := FALSE;
   S702_TL_DC_2ND_CLAMP2.Visu_Adv_Arr[12] := FALSE;
   S702_TL_DC_2ND_CLAMP2.Visu_Adv_Arr[13] := FALSE;
   S702_TL_DC_2ND_CLAMP2.Visu_Adv_Arr[14] := FALSE;
   S702_TL_DC_2ND_CLAMP2.Visu_Adv_Arr[15] := FALSE;
   S702_TL_DC_2ND_CLAMP2.Visu_Ret_Arr[0] := FALSE;
   S702_TL_DC_2ND_CLAMP2.Visu_Ret_Arr[1] := FALSE;
   S702_TL_DC_2ND_CLAMP2.Visu_Ret_Arr[2] := FALSE;
   S702_TL_DC_2ND_CLAMP2.Visu_Ret_Arr[3] := FALSE;
   S702_TL_DC_2ND_CLAMP2.Visu_Ret_Arr[4] := FALSE;
   S702_TL_DC_2ND_CLAMP2.Visu_Ret_Arr[5] := FALSE;
   S702_TL_DC_2ND_CLAMP2.Visu_Ret_Arr[6] := FALSE;
   S702_TL_DC_2ND_CLAMP2.Visu_Ret_Arr[7] := FALSE;
   S702_TL_DC_2ND_CLAMP2.Visu_Ret_Arr[8] := FALSE;
   S702_TL_DC_2ND_CLAMP2.Visu_Ret_Arr[9] := FALSE;
   S702_TL_DC_2ND_CLAMP2.Visu_Ret_Arr[10] := FALSE;
   S702_TL_DC_2ND_CLAMP2.Visu_Ret_Arr[11] := FALSE;
   S702_TL_DC_2ND_CLAMP2.Visu_Ret_Arr[12] := FALSE;
   S702_TL_DC_2ND_CLAMP2.Visu_Ret_Arr[13] := FALSE;
   S702_TL_DC_2ND_CLAMP2.Visu_Ret_Arr[14] := FALSE;
   S702_TL_DC_2ND_CLAMP2.Visu_Ret_Arr[15] := FALSE;
   S702_TL_DC_2ND_CLAMP2.BLK_Move_Ret := 0;
   S702_TL_DC_2ND_CLAMP2.Enable := FALSE;
   S702_TL_DC_2ND_CLAMP2.Adv_End := FALSE;
   S702_TL_DC_2ND_CLAMP2.Ret_End := FALSE;
   S702_TL_DC_U261.Enable_Aux := FALSE;
   S702_TL_DC_U261.Adv_Amount := 0;
   S702_TL_DC_U261.Ret_Amount := 0;
   S702_TL_DC_U261.LS_Adv1 := FALSE;
   S702_TL_DC_U261.LS_Ret1 := FALSE;
   S702_TL_DC_U261.LS_Adv2 := FALSE;
   S702_TL_DC_U261.LS_Ret2 := FALSE;
   S702_TL_DC_U261.LS_Adv3 := FALSE;
   S702_TL_DC_U261.LS_Ret3 := FALSE;
   S702_TL_DC_U261.LS_Adv4 := FALSE;
   S702_TL_DC_U261.LS_Ret4 := FALSE;
   S702_TL_DC_U261.LS_Adv5 := FALSE;
   S702_TL_DC_U261.LS_Ret5 := FALSE;
   S702_TL_DC_U261.LS_Adv6 := FALSE;
   S702_TL_DC_U261.LS_Ret6 := FALSE;
   S702_TL_DC_U261.LS_Adv7 := FALSE;
   S702_TL_DC_U261.LS_Ret7 := FALSE;
   S702_TL_DC_U261.LS_Adv8 := FALSE;
   S702_TL_DC_U261.LS_Ret8 := FALSE;
   S702_TL_DC_U261.SOL_Adv := FALSE;
   S702_TL_DC_U261.SOL_Ret := FALSE;
   S702_TL_DC_U261.M_Ready := FALSE;
   S702_TL_DC_U261.T_CHK1 := T#0MS;
   S702_TL_DC_U261.T_CHK2 := T#0MS;
   S702_TL_DC_U261.PB_Lamp_CHK := FALSE;
   S702_TL_DC_U261.PB_Error_Rst := FALSE;
   S702_TL_DC_U261.M_FLICK := FALSE;
   S702_TL_DC_U261.M_Adv_Err := FALSE;
   S702_TL_DC_U261.M_Ret_Err := FALSE;
   S702_TL_DC_U261.LP_Adv := FALSE;
   S702_TL_DC_U261.LP_Ret := FALSE;
   S702_TL_DC_U261.Visu_Adv := W#16#0;
   S702_TL_DC_U261.Visu_Ret := W#16#0;
   S702_TL_DC_U261.Error_T1.IN := FALSE;
   S702_TL_DC_U261.Error_T1.PT := T#0MS;
   S702_TL_DC_U261.Error_T1.Q := FALSE;
   S702_TL_DC_U261.Error_T1.ET := T#0MS;
   S702_TL_DC_U261.Error_T1.STATE := B#16#0;
   S702_TL_DC_U261.Error_T1.STIME := T#0MS;
   S702_TL_DC_U261.Error_T1.ATIME := T#0MS;
   S702_TL_DC_U261.Error_T2.IN := FALSE;
   S702_TL_DC_U261.Error_T2.PT := T#0MS;
   S702_TL_DC_U261.Error_T2.Q := FALSE;
   S702_TL_DC_U261.Error_T2.ET := T#0MS;
   S702_TL_DC_U261.Error_T2.STATE := B#16#0;
   S702_TL_DC_U261.Error_T2.STIME := T#0MS;
   S702_TL_DC_U261.Error_T2.ATIME := T#0MS;
   S702_TL_DC_U261.Adv_End_Aux := FALSE;
   S702_TL_DC_U261.Ret_End_Aux := FALSE;
   S702_TL_DC_U261.CHK_Aux1 := FALSE;
   S702_TL_DC_U261.CHK_Aux2 := FALSE;
   S702_TL_DC_U261.Error_T1_DN := FALSE;
   S702_TL_DC_U261.Error_T2_DN := FALSE;
   S702_TL_DC_U261.Adv_Memo := FALSE;
   S702_TL_DC_U261.Visu_Adv_Arr[0] := FALSE;
   S702_TL_DC_U261.Visu_Adv_Arr[1] := FALSE;
   S702_TL_DC_U261.Visu_Adv_Arr[2] := FALSE;
   S702_TL_DC_U261.Visu_Adv_Arr[3] := FALSE;
   S702_TL_DC_U261.Visu_Adv_Arr[4] := FALSE;
   S702_TL_DC_U261.Visu_Adv_Arr[5] := FALSE;
   S702_TL_DC_U261.Visu_Adv_Arr[6] := FALSE;
   S702_TL_DC_U261.Visu_Adv_Arr[7] := FALSE;
   S702_TL_DC_U261.Visu_Adv_Arr[8] := FALSE;
   S702_TL_DC_U261.Visu_Adv_Arr[9] := FALSE;
   S702_TL_DC_U261.Visu_Adv_Arr[10] := FALSE;
   S702_TL_DC_U261.Visu_Adv_Arr[11] := FALSE;
   S702_TL_DC_U261.Visu_Adv_Arr[12] := FALSE;
   S702_TL_DC_U261.Visu_Adv_Arr[13] := FALSE;
   S702_TL_DC_U261.Visu_Adv_Arr[14] := FALSE;
   S702_TL_DC_U261.Visu_Adv_Arr[15] := FALSE;
   S702_TL_DC_U261.Visu_Ret_Arr[0] := FALSE;
   S702_TL_DC_U261.Visu_Ret_Arr[1] := FALSE;
   S702_TL_DC_U261.Visu_Ret_Arr[2] := FALSE;
   S702_TL_DC_U261.Visu_Ret_Arr[3] := FALSE;
   S702_TL_DC_U261.Visu_Ret_Arr[4] := FALSE;
   S702_TL_DC_U261.Visu_Ret_Arr[5] := FALSE;
   S702_TL_DC_U261.Visu_Ret_Arr[6] := FALSE;
   S702_TL_DC_U261.Visu_Ret_Arr[7] := FALSE;
   S702_TL_DC_U261.Visu_Ret_Arr[8] := FALSE;
   S702_TL_DC_U261.Visu_Ret_Arr[9] := FALSE;
   S702_TL_DC_U261.Visu_Ret_Arr[10] := FALSE;
   S702_TL_DC_U261.Visu_Ret_Arr[11] := FALSE;
   S702_TL_DC_U261.Visu_Ret_Arr[12] := FALSE;
   S702_TL_DC_U261.Visu_Ret_Arr[13] := FALSE;
   S702_TL_DC_U261.Visu_Ret_Arr[14] := FALSE;
   S702_TL_DC_U261.Visu_Ret_Arr[15] := FALSE;
   S702_TL_DC_U261.BLK_Move_Ret := 0;
   S702_TL_DC_U261.Enable := FALSE;
   S702_TL_DC_U261.Adv_End := FALSE;
   S702_TL_DC_U261.Ret_End := FALSE;
   S702_TL_DC_U261_CLAMP.Enable_Aux := FALSE;
   S702_TL_DC_U261_CLAMP.Adv_Amount := 0;
   S702_TL_DC_U261_CLAMP.Ret_Amount := 0;
   S702_TL_DC_U261_CLAMP.LS_Adv1 := FALSE;
   S702_TL_DC_U261_CLAMP.LS_Ret1 := FALSE;
   S702_TL_DC_U261_CLAMP.LS_Adv2 := FALSE;
   S702_TL_DC_U261_CLAMP.LS_Ret2 := FALSE;
   S702_TL_DC_U261_CLAMP.LS_Adv3 := FALSE;
   S702_TL_DC_U261_CLAMP.LS_Ret3 := FALSE;
   S702_TL_DC_U261_CLAMP.LS_Adv4 := FALSE;
   S702_TL_DC_U261_CLAMP.LS_Ret4 := FALSE;
   S702_TL_DC_U261_CLAMP.LS_Adv5 := FALSE;
   S702_TL_DC_U261_CLAMP.LS_Ret5 := FALSE;
   S702_TL_DC_U261_CLAMP.LS_Adv6 := FALSE;
   S702_TL_DC_U261_CLAMP.LS_Ret6 := FALSE;
   S702_TL_DC_U261_CLAMP.LS_Adv7 := FALSE;
   S702_TL_DC_U261_CLAMP.LS_Ret7 := FALSE;
   S702_TL_DC_U261_CLAMP.LS_Adv8 := FALSE;
   S702_TL_DC_U261_CLAMP.LS_Ret8 := FALSE;
   S702_TL_DC_U261_CLAMP.SOL_Adv := FALSE;
   S702_TL_DC_U261_CLAMP.SOL_Ret := FALSE;
   S702_TL_DC_U261_CLAMP.M_Ready := FALSE;
   S702_TL_DC_U261_CLAMP.T_CHK1 := T#0MS;
   S702_TL_DC_U261_CLAMP.T_CHK2 := T#0MS;
   S702_TL_DC_U261_CLAMP.PB_Lamp_CHK := FALSE;
   S702_TL_DC_U261_CLAMP.PB_Error_Rst := FALSE;
   S702_TL_DC_U261_CLAMP.M_FLICK := FALSE;
   S702_TL_DC_U261_CLAMP.M_Adv_Err := FALSE;
   S702_TL_DC_U261_CLAMP.M_Ret_Err := FALSE;
   S702_TL_DC_U261_CLAMP.LP_Adv := FALSE;
   S702_TL_DC_U261_CLAMP.LP_Ret := FALSE;
   S702_TL_DC_U261_CLAMP.Visu_Adv := W#16#0;
   S702_TL_DC_U261_CLAMP.Visu_Ret := W#16#0;
   S702_TL_DC_U261_CLAMP.Error_T1.IN := FALSE;
   S702_TL_DC_U261_CLAMP.Error_T1.PT := T#0MS;
   S702_TL_DC_U261_CLAMP.Error_T1.Q := FALSE;
   S702_TL_DC_U261_CLAMP.Error_T1.ET := T#0MS;
   S702_TL_DC_U261_CLAMP.Error_T1.STATE := B#16#0;
   S702_TL_DC_U261_CLAMP.Error_T1.STIME := T#0MS;
   S702_TL_DC_U261_CLAMP.Error_T1.ATIME := T#0MS;
   S702_TL_DC_U261_CLAMP.Error_T2.IN := FALSE;
   S702_TL_DC_U261_CLAMP.Error_T2.PT := T#0MS;
   S702_TL_DC_U261_CLAMP.Error_T2.Q := FALSE;
   S702_TL_DC_U261_CLAMP.Error_T2.ET := T#0MS;
   S702_TL_DC_U261_CLAMP.Error_T2.STATE := B#16#0;
   S702_TL_DC_U261_CLAMP.Error_T2.STIME := T#0MS;
   S702_TL_DC_U261_CLAMP.Error_T2.ATIME := T#0MS;
   S702_TL_DC_U261_CLAMP.Adv_End_Aux := FALSE;
   S702_TL_DC_U261_CLAMP.Ret_End_Aux := FALSE;
   S702_TL_DC_U261_CLAMP.CHK_Aux1 := FALSE;
   S702_TL_DC_U261_CLAMP.CHK_Aux2 := FALSE;
   S702_TL_DC_U261_CLAMP.Error_T1_DN := FALSE;
   S702_TL_DC_U261_CLAMP.Error_T2_DN := FALSE;
   S702_TL_DC_U261_CLAMP.Adv_Memo := FALSE;
   S702_TL_DC_U261_CLAMP.Visu_Adv_Arr[0] := FALSE;
   S702_TL_DC_U261_CLAMP.Visu_Adv_Arr[1] := FALSE;
   S702_TL_DC_U261_CLAMP.Visu_Adv_Arr[2] := FALSE;
   S702_TL_DC_U261_CLAMP.Visu_Adv_Arr[3] := FALSE;
   S702_TL_DC_U261_CLAMP.Visu_Adv_Arr[4] := FALSE;
   S702_TL_DC_U261_CLAMP.Visu_Adv_Arr[5] := FALSE;
   S702_TL_DC_U261_CLAMP.Visu_Adv_Arr[6] := FALSE;
   S702_TL_DC_U261_CLAMP.Visu_Adv_Arr[7] := FALSE;
   S702_TL_DC_U261_CLAMP.Visu_Adv_Arr[8] := FALSE;
   S702_TL_DC_U261_CLAMP.Visu_Adv_Arr[9] := FALSE;
   S702_TL_DC_U261_CLAMP.Visu_Adv_Arr[10] := FALSE;
   S702_TL_DC_U261_CLAMP.Visu_Adv_Arr[11] := FALSE;
   S702_TL_DC_U261_CLAMP.Visu_Adv_Arr[12] := FALSE;
   S702_TL_DC_U261_CLAMP.Visu_Adv_Arr[13] := FALSE;
   S702_TL_DC_U261_CLAMP.Visu_Adv_Arr[14] := FALSE;
   S702_TL_DC_U261_CLAMP.Visu_Adv_Arr[15] := FALSE;
   S702_TL_DC_U261_CLAMP.Visu_Ret_Arr[0] := FALSE;
   S702_TL_DC_U261_CLAMP.Visu_Ret_Arr[1] := FALSE;
   S702_TL_DC_U261_CLAMP.Visu_Ret_Arr[2] := FALSE;
   S702_TL_DC_U261_CLAMP.Visu_Ret_Arr[3] := FALSE;
   S702_TL_DC_U261_CLAMP.Visu_Ret_Arr[4] := FALSE;
   S702_TL_DC_U261_CLAMP.Visu_Ret_Arr[5] := FALSE;
   S702_TL_DC_U261_CLAMP.Visu_Ret_Arr[6] := FALSE;
   S702_TL_DC_U261_CLAMP.Visu_Ret_Arr[7] := FALSE;
   S702_TL_DC_U261_CLAMP.Visu_Ret_Arr[8] := FALSE;
   S702_TL_DC_U261_CLAMP.Visu_Ret_Arr[9] := FALSE;
   S702_TL_DC_U261_CLAMP.Visu_Ret_Arr[10] := FALSE;
   S702_TL_DC_U261_CLAMP.Visu_Ret_Arr[11] := FALSE;
   S702_TL_DC_U261_CLAMP.Visu_Ret_Arr[12] := FALSE;
   S702_TL_DC_U261_CLAMP.Visu_Ret_Arr[13] := FALSE;
   S702_TL_DC_U261_CLAMP.Visu_Ret_Arr[14] := FALSE;
   S702_TL_DC_U261_CLAMP.Visu_Ret_Arr[15] := FALSE;
   S702_TL_DC_U261_CLAMP.BLK_Move_Ret := 0;
   S702_TL_DC_U261_CLAMP.Enable := FALSE;
   S702_TL_DC_U261_CLAMP.Adv_End := FALSE;
   S702_TL_DC_U261_CLAMP.Ret_End := FALSE;
   S702_TL_DC_U269.Enable_Aux := FALSE;
   S702_TL_DC_U269.Adv_Amount := 0;
   S702_TL_DC_U269.Ret_Amount := 0;
   S702_TL_DC_U269.LS_Adv1 := FALSE;
   S702_TL_DC_U269.LS_Ret1 := FALSE;
   S702_TL_DC_U269.LS_Adv2 := FALSE;
   S702_TL_DC_U269.LS_Ret2 := FALSE;
   S702_TL_DC_U269.LS_Adv3 := FALSE;
   S702_TL_DC_U269.LS_Ret3 := FALSE;
   S702_TL_DC_U269.LS_Adv4 := FALSE;
   S702_TL_DC_U269.LS_Ret4 := FALSE;
   S702_TL_DC_U269.LS_Adv5 := FALSE;
   S702_TL_DC_U269.LS_Ret5 := FALSE;
   S702_TL_DC_U269.LS_Adv6 := FALSE;
   S702_TL_DC_U269.LS_Ret6 := FALSE;
   S702_TL_DC_U269.LS_Adv7 := FALSE;
   S702_TL_DC_U269.LS_Ret7 := FALSE;
   S702_TL_DC_U269.LS_Adv8 := FALSE;
   S702_TL_DC_U269.LS_Ret8 := FALSE;
   S702_TL_DC_U269.SOL_Adv := FALSE;
   S702_TL_DC_U269.SOL_Ret := FALSE;
   S702_TL_DC_U269.M_Ready := FALSE;
   S702_TL_DC_U269.T_CHK1 := T#0MS;
   S702_TL_DC_U269.T_CHK2 := T#0MS;
   S702_TL_DC_U269.PB_Lamp_CHK := FALSE;
   S702_TL_DC_U269.PB_Error_Rst := FALSE;
   S702_TL_DC_U269.M_FLICK := FALSE;
   S702_TL_DC_U269.M_Adv_Err := FALSE;
   S702_TL_DC_U269.M_Ret_Err := FALSE;
   S702_TL_DC_U269.LP_Adv := FALSE;
   S702_TL_DC_U269.LP_Ret := FALSE;
   S702_TL_DC_U269.Visu_Adv := W#16#0;
   S702_TL_DC_U269.Visu_Ret := W#16#0;
   S702_TL_DC_U269.Error_T1.IN := FALSE;
   S702_TL_DC_U269.Error_T1.PT := T#0MS;
   S702_TL_DC_U269.Error_T1.Q := FALSE;
   S702_TL_DC_U269.Error_T1.ET := T#0MS;
   S702_TL_DC_U269.Error_T1.STATE := B#16#0;
   S702_TL_DC_U269.Error_T1.STIME := T#0MS;
   S702_TL_DC_U269.Error_T1.ATIME := T#0MS;
   S702_TL_DC_U269.Error_T2.IN := FALSE;
   S702_TL_DC_U269.Error_T2.PT := T#0MS;
   S702_TL_DC_U269.Error_T2.Q := FALSE;
   S702_TL_DC_U269.Error_T2.ET := T#0MS;
   S702_TL_DC_U269.Error_T2.STATE := B#16#0;
   S702_TL_DC_U269.Error_T2.STIME := T#0MS;
   S702_TL_DC_U269.Error_T2.ATIME := T#0MS;
   S702_TL_DC_U269.Adv_End_Aux := FALSE;
   S702_TL_DC_U269.Ret_End_Aux := FALSE;
   S702_TL_DC_U269.CHK_Aux1 := FALSE;
   S702_TL_DC_U269.CHK_Aux2 := FALSE;
   S702_TL_DC_U269.Error_T1_DN := FALSE;
   S702_TL_DC_U269.Error_T2_DN := FALSE;
   S702_TL_DC_U269.Adv_Memo := FALSE;
   S702_TL_DC_U269.Visu_Adv_Arr[0] := FALSE;
   S702_TL_DC_U269.Visu_Adv_Arr[1] := FALSE;
   S702_TL_DC_U269.Visu_Adv_Arr[2] := FALSE;
   S702_TL_DC_U269.Visu_Adv_Arr[3] := FALSE;
   S702_TL_DC_U269.Visu_Adv_Arr[4] := FALSE;
   S702_TL_DC_U269.Visu_Adv_Arr[5] := FALSE;
   S702_TL_DC_U269.Visu_Adv_Arr[6] := FALSE;
   S702_TL_DC_U269.Visu_Adv_Arr[7] := FALSE;
   S702_TL_DC_U269.Visu_Adv_Arr[8] := FALSE;
   S702_TL_DC_U269.Visu_Adv_Arr[9] := FALSE;
   S702_TL_DC_U269.Visu_Adv_Arr[10] := FALSE;
   S702_TL_DC_U269.Visu_Adv_Arr[11] := FALSE;
   S702_TL_DC_U269.Visu_Adv_Arr[12] := FALSE;
   S702_TL_DC_U269.Visu_Adv_Arr[13] := FALSE;
   S702_TL_DC_U269.Visu_Adv_Arr[14] := FALSE;
   S702_TL_DC_U269.Visu_Adv_Arr[15] := FALSE;
   S702_TL_DC_U269.Visu_Ret_Arr[0] := FALSE;
   S702_TL_DC_U269.Visu_Ret_Arr[1] := FALSE;
   S702_TL_DC_U269.Visu_Ret_Arr[2] := FALSE;
   S702_TL_DC_U269.Visu_Ret_Arr[3] := FALSE;
   S702_TL_DC_U269.Visu_Ret_Arr[4] := FALSE;
   S702_TL_DC_U269.Visu_Ret_Arr[5] := FALSE;
   S702_TL_DC_U269.Visu_Ret_Arr[6] := FALSE;
   S702_TL_DC_U269.Visu_Ret_Arr[7] := FALSE;
   S702_TL_DC_U269.Visu_Ret_Arr[8] := FALSE;
   S702_TL_DC_U269.Visu_Ret_Arr[9] := FALSE;
   S702_TL_DC_U269.Visu_Ret_Arr[10] := FALSE;
   S702_TL_DC_U269.Visu_Ret_Arr[11] := FALSE;
   S702_TL_DC_U269.Visu_Ret_Arr[12] := FALSE;
   S702_TL_DC_U269.Visu_Ret_Arr[13] := FALSE;
   S702_TL_DC_U269.Visu_Ret_Arr[14] := FALSE;
   S702_TL_DC_U269.Visu_Ret_Arr[15] := FALSE;
   S702_TL_DC_U269.BLK_Move_Ret := 0;
   S702_TL_DC_U269.Enable := FALSE;
   S702_TL_DC_U269.Adv_End := FALSE;
   S702_TL_DC_U269.Ret_End := FALSE;
   S702_TL_DC_U269_CLAMP.Enable_Aux := FALSE;
   S702_TL_DC_U269_CLAMP.Adv_Amount := 0;
   S702_TL_DC_U269_CLAMP.Ret_Amount := 0;
   S702_TL_DC_U269_CLAMP.LS_Adv1 := FALSE;
   S702_TL_DC_U269_CLAMP.LS_Ret1 := FALSE;
   S702_TL_DC_U269_CLAMP.LS_Adv2 := FALSE;
   S702_TL_DC_U269_CLAMP.LS_Ret2 := FALSE;
   S702_TL_DC_U269_CLAMP.LS_Adv3 := FALSE;
   S702_TL_DC_U269_CLAMP.LS_Ret3 := FALSE;
   S702_TL_DC_U269_CLAMP.LS_Adv4 := FALSE;
   S702_TL_DC_U269_CLAMP.LS_Ret4 := FALSE;
   S702_TL_DC_U269_CLAMP.LS_Adv5 := FALSE;
   S702_TL_DC_U269_CLAMP.LS_Ret5 := FALSE;
   S702_TL_DC_U269_CLAMP.LS_Adv6 := FALSE;
   S702_TL_DC_U269_CLAMP.LS_Ret6 := FALSE;
   S702_TL_DC_U269_CLAMP.LS_Adv7 := FALSE;
   S702_TL_DC_U269_CLAMP.LS_Ret7 := FALSE;
   S702_TL_DC_U269_CLAMP.LS_Adv8 := FALSE;
   S702_TL_DC_U269_CLAMP.LS_Ret8 := FALSE;
   S702_TL_DC_U269_CLAMP.SOL_Adv := FALSE;
   S702_TL_DC_U269_CLAMP.SOL_Ret := FALSE;
   S702_TL_DC_U269_CLAMP.M_Ready := FALSE;
   S702_TL_DC_U269_CLAMP.T_CHK1 := T#0MS;
   S702_TL_DC_U269_CLAMP.T_CHK2 := T#0MS;
   S702_TL_DC_U269_CLAMP.PB_Lamp_CHK := FALSE;
   S702_TL_DC_U269_CLAMP.PB_Error_Rst := FALSE;
   S702_TL_DC_U269_CLAMP.M_FLICK := FALSE;
   S702_TL_DC_U269_CLAMP.M_Adv_Err := FALSE;
   S702_TL_DC_U269_CLAMP.M_Ret_Err := FALSE;
   S702_TL_DC_U269_CLAMP.LP_Adv := FALSE;
   S702_TL_DC_U269_CLAMP.LP_Ret := FALSE;
   S702_TL_DC_U269_CLAMP.Visu_Adv := W#16#0;
   S702_TL_DC_U269_CLAMP.Visu_Ret := W#16#0;
   S702_TL_DC_U269_CLAMP.Error_T1.IN := FALSE;
   S702_TL_DC_U269_CLAMP.Error_T1.PT := T#0MS;
   S702_TL_DC_U269_CLAMP.Error_T1.Q := FALSE;
   S702_TL_DC_U269_CLAMP.Error_T1.ET := T#0MS;
   S702_TL_DC_U269_CLAMP.Error_T1.STATE := B#16#0;
   S702_TL_DC_U269_CLAMP.Error_T1.STIME := T#0MS;
   S702_TL_DC_U269_CLAMP.Error_T1.ATIME := T#0MS;
   S702_TL_DC_U269_CLAMP.Error_T2.IN := FALSE;
   S702_TL_DC_U269_CLAMP.Error_T2.PT := T#0MS;
   S702_TL_DC_U269_CLAMP.Error_T2.Q := FALSE;
   S702_TL_DC_U269_CLAMP.Error_T2.ET := T#0MS;
   S702_TL_DC_U269_CLAMP.Error_T2.STATE := B#16#0;
   S702_TL_DC_U269_CLAMP.Error_T2.STIME := T#0MS;
   S702_TL_DC_U269_CLAMP.Error_T2.ATIME := T#0MS;
   S702_TL_DC_U269_CLAMP.Adv_End_Aux := FALSE;
   S702_TL_DC_U269_CLAMP.Ret_End_Aux := FALSE;
   S702_TL_DC_U269_CLAMP.CHK_Aux1 := FALSE;
   S702_TL_DC_U269_CLAMP.CHK_Aux2 := FALSE;
   S702_TL_DC_U269_CLAMP.Error_T1_DN := FALSE;
   S702_TL_DC_U269_CLAMP.Error_T2_DN := FALSE;
   S702_TL_DC_U269_CLAMP.Adv_Memo := FALSE;
   S702_TL_DC_U269_CLAMP.Visu_Adv_Arr[0] := FALSE;
   S702_TL_DC_U269_CLAMP.Visu_Adv_Arr[1] := FALSE;
   S702_TL_DC_U269_CLAMP.Visu_Adv_Arr[2] := FALSE;
   S702_TL_DC_U269_CLAMP.Visu_Adv_Arr[3] := FALSE;
   S702_TL_DC_U269_CLAMP.Visu_Adv_Arr[4] := FALSE;
   S702_TL_DC_U269_CLAMP.Visu_Adv_Arr[5] := FALSE;
   S702_TL_DC_U269_CLAMP.Visu_Adv_Arr[6] := FALSE;
   S702_TL_DC_U269_CLAMP.Visu_Adv_Arr[7] := FALSE;
   S702_TL_DC_U269_CLAMP.Visu_Adv_Arr[8] := FALSE;
   S702_TL_DC_U269_CLAMP.Visu_Adv_Arr[9] := FALSE;
   S702_TL_DC_U269_CLAMP.Visu_Adv_Arr[10] := FALSE;
   S702_TL_DC_U269_CLAMP.Visu_Adv_Arr[11] := FALSE;
   S702_TL_DC_U269_CLAMP.Visu_Adv_Arr[12] := FALSE;
   S702_TL_DC_U269_CLAMP.Visu_Adv_Arr[13] := FALSE;
   S702_TL_DC_U269_CLAMP.Visu_Adv_Arr[14] := FALSE;
   S702_TL_DC_U269_CLAMP.Visu_Adv_Arr[15] := FALSE;
   S702_TL_DC_U269_CLAMP.Visu_Ret_Arr[0] := FALSE;
   S702_TL_DC_U269_CLAMP.Visu_Ret_Arr[1] := FALSE;
   S702_TL_DC_U269_CLAMP.Visu_Ret_Arr[2] := FALSE;
   S702_TL_DC_U269_CLAMP.Visu_Ret_Arr[3] := FALSE;
   S702_TL_DC_U269_CLAMP.Visu_Ret_Arr[4] := FALSE;
   S702_TL_DC_U269_CLAMP.Visu_Ret_Arr[5] := FALSE;
   S702_TL_DC_U269_CLAMP.Visu_Ret_Arr[6] := FALSE;
   S702_TL_DC_U269_CLAMP.Visu_Ret_Arr[7] := FALSE;
   S702_TL_DC_U269_CLAMP.Visu_Ret_Arr[8] := FALSE;
   S702_TL_DC_U269_CLAMP.Visu_Ret_Arr[9] := FALSE;
   S702_TL_DC_U269_CLAMP.Visu_Ret_Arr[10] := FALSE;
   S702_TL_DC_U269_CLAMP.Visu_Ret_Arr[11] := FALSE;
   S702_TL_DC_U269_CLAMP.Visu_Ret_Arr[12] := FALSE;
   S702_TL_DC_U269_CLAMP.Visu_Ret_Arr[13] := FALSE;
   S702_TL_DC_U269_CLAMP.Visu_Ret_Arr[14] := FALSE;
   S702_TL_DC_U269_CLAMP.Visu_Ret_Arr[15] := FALSE;
   S702_TL_DC_U269_CLAMP.BLK_Move_Ret := 0;
   S702_TL_DC_U269_CLAMP.Enable := FALSE;
   S702_TL_DC_U269_CLAMP.Adv_End := FALSE;
   S702_TL_DC_U269_CLAMP.Ret_End := FALSE;
   S702_TL_DC_3RD_CLAMP.Enable_Aux := FALSE;
   S702_TL_DC_3RD_CLAMP.Adv_Amount := 0;
   S702_TL_DC_3RD_CLAMP.Ret_Amount := 0;
   S702_TL_DC_3RD_CLAMP.LS_Adv1 := FALSE;
   S702_TL_DC_3RD_CLAMP.LS_Ret1 := FALSE;
   S702_TL_DC_3RD_CLAMP.LS_Adv2 := FALSE;
   S702_TL_DC_3RD_CLAMP.LS_Ret2 := FALSE;
   S702_TL_DC_3RD_CLAMP.LS_Adv3 := FALSE;
   S702_TL_DC_3RD_CLAMP.LS_Ret3 := FALSE;
   S702_TL_DC_3RD_CLAMP.LS_Adv4 := FALSE;
   S702_TL_DC_3RD_CLAMP.LS_Ret4 := FALSE;
   S702_TL_DC_3RD_CLAMP.LS_Adv5 := FALSE;
   S702_TL_DC_3RD_CLAMP.LS_Ret5 := FALSE;
   S702_TL_DC_3RD_CLAMP.LS_Adv6 := FALSE;
   S702_TL_DC_3RD_CLAMP.LS_Ret6 := FALSE;
   S702_TL_DC_3RD_CLAMP.LS_Adv7 := FALSE;
   S702_TL_DC_3RD_CLAMP.LS_Ret7 := FALSE;
   S702_TL_DC_3RD_CLAMP.LS_Adv8 := FALSE;
   S702_TL_DC_3RD_CLAMP.LS_Ret8 := FALSE;
   S702_TL_DC_3RD_CLAMP.SOL_Adv := FALSE;
   S702_TL_DC_3RD_CLAMP.SOL_Ret := FALSE;
   S702_TL_DC_3RD_CLAMP.M_Ready := FALSE;
   S702_TL_DC_3RD_CLAMP.T_CHK1 := T#0MS;
   S702_TL_DC_3RD_CLAMP.T_CHK2 := T#0MS;
   S702_TL_DC_3RD_CLAMP.PB_Lamp_CHK := FALSE;
   S702_TL_DC_3RD_CLAMP.PB_Error_Rst := FALSE;
   S702_TL_DC_3RD_CLAMP.M_FLICK := FALSE;
   S702_TL_DC_3RD_CLAMP.M_Adv_Err := FALSE;
   S702_TL_DC_3RD_CLAMP.M_Ret_Err := FALSE;
   S702_TL_DC_3RD_CLAMP.LP_Adv := FALSE;
   S702_TL_DC_3RD_CLAMP.LP_Ret := FALSE;
   S702_TL_DC_3RD_CLAMP.Visu_Adv := W#16#0;
   S702_TL_DC_3RD_CLAMP.Visu_Ret := W#16#0;
   S702_TL_DC_3RD_CLAMP.Error_T1.IN := FALSE;
   S702_TL_DC_3RD_CLAMP.Error_T1.PT := T#0MS;
   S702_TL_DC_3RD_CLAMP.Error_T1.Q := FALSE;
   S702_TL_DC_3RD_CLAMP.Error_T1.ET := T#0MS;
   S702_TL_DC_3RD_CLAMP.Error_T1.STATE := B#16#0;
   S702_TL_DC_3RD_CLAMP.Error_T1.STIME := T#0MS;
   S702_TL_DC_3RD_CLAMP.Error_T1.ATIME := T#0MS;
   S702_TL_DC_3RD_CLAMP.Error_T2.IN := FALSE;
   S702_TL_DC_3RD_CLAMP.Error_T2.PT := T#0MS;
   S702_TL_DC_3RD_CLAMP.Error_T2.Q := FALSE;
   S702_TL_DC_3RD_CLAMP.Error_T2.ET := T#0MS;
   S702_TL_DC_3RD_CLAMP.Error_T2.STATE := B#16#0;
   S702_TL_DC_3RD_CLAMP.Error_T2.STIME := T#0MS;
   S702_TL_DC_3RD_CLAMP.Error_T2.ATIME := T#0MS;
   S702_TL_DC_3RD_CLAMP.Adv_End_Aux := FALSE;
   S702_TL_DC_3RD_CLAMP.Ret_End_Aux := FALSE;
   S702_TL_DC_3RD_CLAMP.CHK_Aux1 := FALSE;
   S702_TL_DC_3RD_CLAMP.CHK_Aux2 := FALSE;
   S702_TL_DC_3RD_CLAMP.Error_T1_DN := FALSE;
   S702_TL_DC_3RD_CLAMP.Error_T2_DN := FALSE;
   S702_TL_DC_3RD_CLAMP.Adv_Memo := FALSE;
   S702_TL_DC_3RD_CLAMP.Visu_Adv_Arr[0] := FALSE;
   S702_TL_DC_3RD_CLAMP.Visu_Adv_Arr[1] := FALSE;
   S702_TL_DC_3RD_CLAMP.Visu_Adv_Arr[2] := FALSE;
   S702_TL_DC_3RD_CLAMP.Visu_Adv_Arr[3] := FALSE;
   S702_TL_DC_3RD_CLAMP.Visu_Adv_Arr[4] := FALSE;
   S702_TL_DC_3RD_CLAMP.Visu_Adv_Arr[5] := FALSE;
   S702_TL_DC_3RD_CLAMP.Visu_Adv_Arr[6] := FALSE;
   S702_TL_DC_3RD_CLAMP.Visu_Adv_Arr[7] := FALSE;
   S702_TL_DC_3RD_CLAMP.Visu_Adv_Arr[8] := FALSE;
   S702_TL_DC_3RD_CLAMP.Visu_Adv_Arr[9] := FALSE;
   S702_TL_DC_3RD_CLAMP.Visu_Adv_Arr[10] := FALSE;
   S702_TL_DC_3RD_CLAMP.Visu_Adv_Arr[11] := FALSE;
   S702_TL_DC_3RD_CLAMP.Visu_Adv_Arr[12] := FALSE;
   S702_TL_DC_3RD_CLAMP.Visu_Adv_Arr[13] := FALSE;
   S702_TL_DC_3RD_CLAMP.Visu_Adv_Arr[14] := FALSE;
   S702_TL_DC_3RD_CLAMP.Visu_Adv_Arr[15] := FALSE;
   S702_TL_DC_3RD_CLAMP.Visu_Ret_Arr[0] := FALSE;
   S702_TL_DC_3RD_CLAMP.Visu_Ret_Arr[1] := FALSE;
   S702_TL_DC_3RD_CLAMP.Visu_Ret_Arr[2] := FALSE;
   S702_TL_DC_3RD_CLAMP.Visu_Ret_Arr[3] := FALSE;
   S702_TL_DC_3RD_CLAMP.Visu_Ret_Arr[4] := FALSE;
   S702_TL_DC_3RD_CLAMP.Visu_Ret_Arr[5] := FALSE;
   S702_TL_DC_3RD_CLAMP.Visu_Ret_Arr[6] := FALSE;
   S702_TL_DC_3RD_CLAMP.Visu_Ret_Arr[7] := FALSE;
   S702_TL_DC_3RD_CLAMP.Visu_Ret_Arr[8] := FALSE;
   S702_TL_DC_3RD_CLAMP.Visu_Ret_Arr[9] := FALSE;
   S702_TL_DC_3RD_CLAMP.Visu_Ret_Arr[10] := FALSE;
   S702_TL_DC_3RD_CLAMP.Visu_Ret_Arr[11] := FALSE;
   S702_TL_DC_3RD_CLAMP.Visu_Ret_Arr[12] := FALSE;
   S702_TL_DC_3RD_CLAMP.Visu_Ret_Arr[13] := FALSE;
   S702_TL_DC_3RD_CLAMP.Visu_Ret_Arr[14] := FALSE;
   S702_TL_DC_3RD_CLAMP.Visu_Ret_Arr[15] := FALSE;
   S702_TL_DC_3RD_CLAMP.BLK_Move_Ret := 0;
   S702_TL_DC_3RD_CLAMP.Enable := FALSE;
   S702_TL_DC_3RD_CLAMP.Adv_End := FALSE;
   S702_TL_DC_3RD_CLAMP.Ret_End := FALSE;
   S702_TL_DC_U262_1_UP_DN.Enable_Aux := FALSE;
   S702_TL_DC_U262_1_UP_DN.Adv_Amount := 0;
   S702_TL_DC_U262_1_UP_DN.Ret_Amount := 0;
   S702_TL_DC_U262_1_UP_DN.LS_Adv1 := FALSE;
   S702_TL_DC_U262_1_UP_DN.LS_Ret1 := FALSE;
   S702_TL_DC_U262_1_UP_DN.LS_Adv2 := FALSE;
   S702_TL_DC_U262_1_UP_DN.LS_Ret2 := FALSE;
   S702_TL_DC_U262_1_UP_DN.LS_Adv3 := FALSE;
   S702_TL_DC_U262_1_UP_DN.LS_Ret3 := FALSE;
   S702_TL_DC_U262_1_UP_DN.LS_Adv4 := FALSE;
   S702_TL_DC_U262_1_UP_DN.LS_Ret4 := FALSE;
   S702_TL_DC_U262_1_UP_DN.LS_Adv5 := FALSE;
   S702_TL_DC_U262_1_UP_DN.LS_Ret5 := FALSE;
   S702_TL_DC_U262_1_UP_DN.LS_Adv6 := FALSE;
   S702_TL_DC_U262_1_UP_DN.LS_Ret6 := FALSE;
   S702_TL_DC_U262_1_UP_DN.LS_Adv7 := FALSE;
   S702_TL_DC_U262_1_UP_DN.LS_Ret7 := FALSE;
   S702_TL_DC_U262_1_UP_DN.LS_Adv8 := FALSE;
   S702_TL_DC_U262_1_UP_DN.LS_Ret8 := FALSE;
   S702_TL_DC_U262_1_UP_DN.SOL_Adv := FALSE;
   S702_TL_DC_U262_1_UP_DN.SOL_Ret := FALSE;
   S702_TL_DC_U262_1_UP_DN.M_Ready := FALSE;
   S702_TL_DC_U262_1_UP_DN.T_CHK1 := T#0MS;
   S702_TL_DC_U262_1_UP_DN.T_CHK2 := T#0MS;
   S702_TL_DC_U262_1_UP_DN.PB_Lamp_CHK := FALSE;
   S702_TL_DC_U262_1_UP_DN.PB_Error_Rst := FALSE;
   S702_TL_DC_U262_1_UP_DN.M_FLICK := FALSE;
   S702_TL_DC_U262_1_UP_DN.M_Adv_Err := FALSE;
   S702_TL_DC_U262_1_UP_DN.M_Ret_Err := FALSE;
   S702_TL_DC_U262_1_UP_DN.LP_Adv := FALSE;
   S702_TL_DC_U262_1_UP_DN.LP_Ret := FALSE;
   S702_TL_DC_U262_1_UP_DN.Visu_Adv := W#16#0;
   S702_TL_DC_U262_1_UP_DN.Visu_Ret := W#16#0;
   S702_TL_DC_U262_1_UP_DN.Error_T1.IN := FALSE;
   S702_TL_DC_U262_1_UP_DN.Error_T1.PT := T#0MS;
   S702_TL_DC_U262_1_UP_DN.Error_T1.Q := FALSE;
   S702_TL_DC_U262_1_UP_DN.Error_T1.ET := T#0MS;
   S702_TL_DC_U262_1_UP_DN.Error_T1.STATE := B#16#0;
   S702_TL_DC_U262_1_UP_DN.Error_T1.STIME := T#0MS;
   S702_TL_DC_U262_1_UP_DN.Error_T1.ATIME := T#0MS;
   S702_TL_DC_U262_1_UP_DN.Error_T2.IN := FALSE;
   S702_TL_DC_U262_1_UP_DN.Error_T2.PT := T#0MS;
   S702_TL_DC_U262_1_UP_DN.Error_T2.Q := FALSE;
   S702_TL_DC_U262_1_UP_DN.Error_T2.ET := T#0MS;
   S702_TL_DC_U262_1_UP_DN.Error_T2.STATE := B#16#0;
   S702_TL_DC_U262_1_UP_DN.Error_T2.STIME := T#0MS;
   S702_TL_DC_U262_1_UP_DN.Error_T2.ATIME := T#0MS;
   S702_TL_DC_U262_1_UP_DN.Adv_End_Aux := FALSE;
   S702_TL_DC_U262_1_UP_DN.Ret_End_Aux := FALSE;
   S702_TL_DC_U262_1_UP_DN.CHK_Aux1 := FALSE;
   S702_TL_DC_U262_1_UP_DN.CHK_Aux2 := FALSE;
   S702_TL_DC_U262_1_UP_DN.Error_T1_DN := FALSE;
   S702_TL_DC_U262_1_UP_DN.Error_T2_DN := FALSE;
   S702_TL_DC_U262_1_UP_DN.Adv_Memo := FALSE;
   S702_TL_DC_U262_1_UP_DN.Visu_Adv_Arr[0] := FALSE;
   S702_TL_DC_U262_1_UP_DN.Visu_Adv_Arr[1] := FALSE;
   S702_TL_DC_U262_1_UP_DN.Visu_Adv_Arr[2] := FALSE;
   S702_TL_DC_U262_1_UP_DN.Visu_Adv_Arr[3] := FALSE;
   S702_TL_DC_U262_1_UP_DN.Visu_Adv_Arr[4] := FALSE;
   S702_TL_DC_U262_1_UP_DN.Visu_Adv_Arr[5] := FALSE;
   S702_TL_DC_U262_1_UP_DN.Visu_Adv_Arr[6] := FALSE;
   S702_TL_DC_U262_1_UP_DN.Visu_Adv_Arr[7] := FALSE;
   S702_TL_DC_U262_1_UP_DN.Visu_Adv_Arr[8] := FALSE;
   S702_TL_DC_U262_1_UP_DN.Visu_Adv_Arr[9] := FALSE;
   S702_TL_DC_U262_1_UP_DN.Visu_Adv_Arr[10] := FALSE;
   S702_TL_DC_U262_1_UP_DN.Visu_Adv_Arr[11] := FALSE;
   S702_TL_DC_U262_1_UP_DN.Visu_Adv_Arr[12] := FALSE;
   S702_TL_DC_U262_1_UP_DN.Visu_Adv_Arr[13] := FALSE;
   S702_TL_DC_U262_1_UP_DN.Visu_Adv_Arr[14] := FALSE;
   S702_TL_DC_U262_1_UP_DN.Visu_Adv_Arr[15] := FALSE;
   S702_TL_DC_U262_1_UP_DN.Visu_Ret_Arr[0] := FALSE;
   S702_TL_DC_U262_1_UP_DN.Visu_Ret_Arr[1] := FALSE;
   S702_TL_DC_U262_1_UP_DN.Visu_Ret_Arr[2] := FALSE;
   S702_TL_DC_U262_1_UP_DN.Visu_Ret_Arr[3] := FALSE;
   S702_TL_DC_U262_1_UP_DN.Visu_Ret_Arr[4] := FALSE;
   S702_TL_DC_U262_1_UP_DN.Visu_Ret_Arr[5] := FALSE;
   S702_TL_DC_U262_1_UP_DN.Visu_Ret_Arr[6] := FALSE;
   S702_TL_DC_U262_1_UP_DN.Visu_Ret_Arr[7] := FALSE;
   S702_TL_DC_U262_1_UP_DN.Visu_Ret_Arr[8] := FALSE;
   S702_TL_DC_U262_1_UP_DN.Visu_Ret_Arr[9] := FALSE;
   S702_TL_DC_U262_1_UP_DN.Visu_Ret_Arr[10] := FALSE;
   S702_TL_DC_U262_1_UP_DN.Visu_Ret_Arr[11] := FALSE;
   S702_TL_DC_U262_1_UP_DN.Visu_Ret_Arr[12] := FALSE;
   S702_TL_DC_U262_1_UP_DN.Visu_Ret_Arr[13] := FALSE;
   S702_TL_DC_U262_1_UP_DN.Visu_Ret_Arr[14] := FALSE;
   S702_TL_DC_U262_1_UP_DN.Visu_Ret_Arr[15] := FALSE;
   S702_TL_DC_U262_1_UP_DN.BLK_Move_Ret := 0;
   S702_TL_DC_U262_1_UP_DN.Enable := FALSE;
   S702_TL_DC_U262_1_UP_DN.Adv_End := FALSE;
   S702_TL_DC_U262_1_UP_DN.Ret_End := FALSE;
   S702_TL_DC_U262_1.Enable_Aux := FALSE;
   S702_TL_DC_U262_1.Adv_Amount := 0;
   S702_TL_DC_U262_1.Ret_Amount := 0;
   S702_TL_DC_U262_1.LS_Adv1 := FALSE;
   S702_TL_DC_U262_1.LS_Ret1 := FALSE;
   S702_TL_DC_U262_1.LS_Adv2 := FALSE;
   S702_TL_DC_U262_1.LS_Ret2 := FALSE;
   S702_TL_DC_U262_1.LS_Adv3 := FALSE;
   S702_TL_DC_U262_1.LS_Ret3 := FALSE;
   S702_TL_DC_U262_1.LS_Adv4 := FALSE;
   S702_TL_DC_U262_1.LS_Ret4 := FALSE;
   S702_TL_DC_U262_1.LS_Adv5 := FALSE;
   S702_TL_DC_U262_1.LS_Ret5 := FALSE;
   S702_TL_DC_U262_1.LS_Adv6 := FALSE;
   S702_TL_DC_U262_1.LS_Ret6 := FALSE;
   S702_TL_DC_U262_1.LS_Adv7 := FALSE;
   S702_TL_DC_U262_1.LS_Ret7 := FALSE;
   S702_TL_DC_U262_1.LS_Adv8 := FALSE;
   S702_TL_DC_U262_1.LS_Ret8 := FALSE;
   S702_TL_DC_U262_1.SOL_Adv := FALSE;
   S702_TL_DC_U262_1.SOL_Ret := FALSE;
   S702_TL_DC_U262_1.M_Ready := FALSE;
   S702_TL_DC_U262_1.T_CHK1 := T#0MS;
   S702_TL_DC_U262_1.T_CHK2 := T#0MS;
   S702_TL_DC_U262_1.PB_Lamp_CHK := FALSE;
   S702_TL_DC_U262_1.PB_Error_Rst := FALSE;
   S702_TL_DC_U262_1.M_FLICK := FALSE;
   S702_TL_DC_U262_1.M_Adv_Err := FALSE;
   S702_TL_DC_U262_1.M_Ret_Err := FALSE;
   S702_TL_DC_U262_1.LP_Adv := FALSE;
   S702_TL_DC_U262_1.LP_Ret := FALSE;
   S702_TL_DC_U262_1.Visu_Adv := W#16#0;
   S702_TL_DC_U262_1.Visu_Ret := W#16#0;
   S702_TL_DC_U262_1.Error_T1.IN := FALSE;
   S702_TL_DC_U262_1.Error_T1.PT := T#0MS;
   S702_TL_DC_U262_1.Error_T1.Q := FALSE;
   S702_TL_DC_U262_1.Error_T1.ET := T#0MS;
   S702_TL_DC_U262_1.Error_T1.STATE := B#16#0;
   S702_TL_DC_U262_1.Error_T1.STIME := T#0MS;
   S702_TL_DC_U262_1.Error_T1.ATIME := T#0MS;
   S702_TL_DC_U262_1.Error_T2.IN := FALSE;
   S702_TL_DC_U262_1.Error_T2.PT := T#0MS;
   S702_TL_DC_U262_1.Error_T2.Q := FALSE;
   S702_TL_DC_U262_1.Error_T2.ET := T#0MS;
   S702_TL_DC_U262_1.Error_T2.STATE := B#16#0;
   S702_TL_DC_U262_1.Error_T2.STIME := T#0MS;
   S702_TL_DC_U262_1.Error_T2.ATIME := T#0MS;
   S702_TL_DC_U262_1.Adv_End_Aux := FALSE;
   S702_TL_DC_U262_1.Ret_End_Aux := FALSE;
   S702_TL_DC_U262_1.CHK_Aux1 := FALSE;
   S702_TL_DC_U262_1.CHK_Aux2 := FALSE;
   S702_TL_DC_U262_1.Error_T1_DN := FALSE;
   S702_TL_DC_U262_1.Error_T2_DN := FALSE;
   S702_TL_DC_U262_1.Adv_Memo := FALSE;
   S702_TL_DC_U262_1.Visu_Adv_Arr[0] := FALSE;
   S702_TL_DC_U262_1.Visu_Adv_Arr[1] := FALSE;
   S702_TL_DC_U262_1.Visu_Adv_Arr[2] := FALSE;
   S702_TL_DC_U262_1.Visu_Adv_Arr[3] := FALSE;
   S702_TL_DC_U262_1.Visu_Adv_Arr[4] := FALSE;
   S702_TL_DC_U262_1.Visu_Adv_Arr[5] := FALSE;
   S702_TL_DC_U262_1.Visu_Adv_Arr[6] := FALSE;
   S702_TL_DC_U262_1.Visu_Adv_Arr[7] := FALSE;
   S702_TL_DC_U262_1.Visu_Adv_Arr[8] := FALSE;
   S702_TL_DC_U262_1.Visu_Adv_Arr[9] := FALSE;
   S702_TL_DC_U262_1.Visu_Adv_Arr[10] := FALSE;
   S702_TL_DC_U262_1.Visu_Adv_Arr[11] := FALSE;
   S702_TL_DC_U262_1.Visu_Adv_Arr[12] := FALSE;
   S702_TL_DC_U262_1.Visu_Adv_Arr[13] := FALSE;
